// TwinCAT 3 PLC project ValentaDCmotor
// ProgramVersion: 3.1.4026.20
// libraries:
//   Tc2_Standard, * (Beckhoff Automation GmbH)
//   Tc2_System, * (Beckhoff Automation GmbH)
//   Tc3_Module, * (Beckhoff Automation GmbH)
//   VisuDialogs, * (System)
//   VisuSymbols,3.5.10.0,System
// project tree:
//   DUTs/ E_Color.TcDUT, E_ControlMode.TcDUT, E_DoorState.TcDUT, ST_KeyControl.TcDUT, E_BlinkMarine_Color.TcDUT, E_GearState.TcDUT, E_LedColor.TcDUT, E_BacklightColor.TcDUT, E_ValveState.TcDUT, ST_UcWinchControl.TcDUT
//   / GlobalTextList.TcGTLO, PlcTask.TcTTO
//   GVLs/ GVL.TcGVL, GVL_Alarms.TcGVL, GVL_CAN.TcGVL, GVL_ENGINE.TcGVL, GVL_HMI.TcGVL, GVL_IO.TcGVL, GVL_PERSISTENT.TcGVL
//   POUs/ DirectMotorControl.TcPOU, MAIN.TcPOU, PRG_Ballast.TcPOU, PRG_BlinkMarine.TcPOU, PRG_Doors.TcPOU, PRG_Engine.TcPOU, PRG_HmiLeds.TcPOU, PRG_Sequence.TcPOU, PRG_StationManager.TcPOU, PRG_Can.TcPOU, PRG_Winches.TcPOU, PRG_ZF_Control.TcPOU
//   POUs/FBs/ FB_BallastValve.TcPOU, FB_DC_Motor_Direct_Ctrl.TcPOU, FB_DoorControl.TcPOU, FB_EngineControl.TcPOU, FB_StationManager.TcPOU, FB_TankScaling.TcPOU, FB_TunelPump.TcPOU, FB_WinchControl.TcPOU, MeasureRPM.TcPOU
//   POUs/Sim/ E_SystemMode.TcDUT, PRG_SimDoors.TcPOU
//   VISUs/ Visualization1.TcVIS, Visualization2.TcVIS, VisualizationManager.TcVMO (not stored), VisuDoorControl.TcVIS
// real-time tasks:
//   TASK PlcTask: cycle T#2ms, priority 20, ADS port 350
// I/O:
//   DEVICE Device 1 (EtherCAT), AmsNetId 5.168.36.149.2.1
//     Term 1 (EK1200) [EK1200-5000 EtherCAT Power supply (2A E-Bus)]
//       Term 2 (EL1008) [EL1008 8Ch. Dig. Input 24V, 3ms]
//       Term 3 (EL2008) [EL2008 8Ch. Dig. Output 24V, 0.5A]
//       Term 4 (EL4018) [EL4018 8Ch. Ana. Output 0-20mA, 12bit]
//       Term 5 (EL6751) [EL6751 CANopen Master]
//       Term 6 (EK1110) [EK1110 EtherCAT extension]
//     Term 7 (EK1100) [EK1100 EtherCAT Coupler (2A E-Bus)]
//       Term 8 (EL1008) [EL1008 8Ch. Dig. Input 24V, 3ms]
//       Term 9 (EL1008) [EL1008 8Ch. Dig. Input 24V, 3ms]
//       Term 10 (EL1008) [EL1008 8Ch. Dig. Input 24V, 3ms]
//       Term 11 (EL3014) [EL3014 4Ch. Ana. Input 0-20mA DIFF]
//       Term 12 (EL3014) [EL3014 4Ch. Ana. Input 0-20mA DIFF]
//       Term 13 (EL3014) [EL3014 4Ch. Ana. Input 0-20mA DIFF]
//       Term 14 (EL3004) [EL3004 4Ch. Ana. Input +/-10V]
//       Term 15 (EL3255) [EL3255 5Ch. potentiometer measurement with sensor supply]
//       Term 16 (EL7342) [EL7342 2Ch. DC motor output stage (50V, 3.5A)]
//       Term 17 (EL2008) [EL2008 8Ch. Dig. Output 24V, 0.5A]
//       Term 18 (EL2008) [EL2008 8Ch. Dig. Output 24V, 0.5A]
//       Term 19 (EL2008) [EL2008 8Ch. Dig. Output 24V, 0.5A]
//       Term 20 (EL2008) [EL2008 8Ch. Dig. Output 24V, 0.5A]
//       Term 21 (EL9011) [EL9011 End Terminal]
//   DEVICE Device 2 (EL6751), AmsNetId 5.168.36.149.3.1
//     Box 10 (BlinkMarine)
//     Box 11 (BlinkMarine)
//     Box 20 (BlinkMarine)
// variable links:
//   ValentaDCmotor/ValentaDCmotor Instance <-> Device 1 (EtherCAT)/Term 7 (EK1100)/Term 15 (EL3255)
//     PlcTask Inputs/GVL.iwPotFeedback_M1 <-> AI Standard Channel 1/Value
//     PlcTask Inputs/GVL.iwPotFeedback_M2 <-> AI Standard Channel 2/Value
//     PlcTask Inputs/GVL_IO.iLever_St1_Raw <-> AI Standard Channel 3/Value
//     PlcTask Inputs/GVL_IO.iLever_St2_Raw <-> AI Standard Channel 4/Value
//   ValentaDCmotor/ValentaDCmotor Instance <-> Device 1 (EtherCAT)/Term 7 (EK1100)/Term 16 (EL7342)
//     PlcTask Inputs/GVL.bDigitalInput1_M1 <-> DCM Status Channel 1/Status/Digital input 1
//     PlcTask Inputs/GVL.bDigitalInput1_M2 <-> DCM Status Channel 2/Status/Digital input 1
//     PlcTask Inputs/GVL.bDigitalInput2_M1 <-> DCM Status Channel 1/Status/Digital input 2
//     PlcTask Inputs/GVL.bDigitalInput2_M2 <-> DCM Status Channel 2/Status/Digital input 2
//     PlcTask Inputs/GVL.bError_M1 <-> DCM Status Channel 1/Status/Error
//     PlcTask Inputs/GVL.bError_M2 <-> DCM Status Channel 2/Status/Error
//     PlcTask Inputs/GVL.bMovingNegative_M1 <-> DCM Status Channel 1/Status/Moving negative
//     PlcTask Inputs/GVL.bMovingNegative_M2 <-> DCM Status Channel 2/Status/Moving negative
//     PlcTask Inputs/GVL.bMovingPositive_M1 <-> DCM Status Channel 1/Status/Moving positive
//     PlcTask Inputs/GVL.bMovingPositive_M2 <-> DCM Status Channel 2/Status/Moving positive
//     PlcTask Inputs/GVL.bReadyToEnable_M1 <-> DCM Status Channel 1/Status/Ready to enable
//     PlcTask Inputs/GVL.bReadyToEnable_M2 <-> DCM Status Channel 2/Status/Ready to enable
//     PlcTask Inputs/GVL.bReady_M1 <-> DCM Status Channel 1/Status/Ready
//     PlcTask Inputs/GVL.bReady_M2 <-> DCM Status Channel 2/Status/Ready
//     PlcTask Inputs/GVL.bSyncError_M1 <-> DCM Status Channel 1/Status/Sync error
//     PlcTask Inputs/GVL.bSyncError_M2 <-> DCM Status Channel 2/Status/Sync error
//     PlcTask Inputs/GVL.bTorqueReduced_M1 <-> DCM Status Channel 1/Status/Torque reduced
//     PlcTask Inputs/GVL.bTorqueReduced_M2 <-> DCM Status Channel 2/Status/Torque reduced
//     PlcTask Inputs/GVL.bTxPDOToggle_M1 <-> DCM Status Channel 1/Status/TxPDO Toggle
//     PlcTask Inputs/GVL.bTxPDOToggle_M2 <-> DCM Status Channel 2/Status/TxPDO Toggle
//     PlcTask Inputs/GVL.bWarning_M1 <-> DCM Status Channel 1/Status/Warning
//     PlcTask Inputs/GVL.bWarning_M2 <-> DCM Status Channel 2/Status/Warning
//     PlcTask Inputs/GVL.nMotorCurrent_M1 <-> DCM Synchron info data Channel 1/Info data 2
//     PlcTask Inputs/GVL.nMotorCurrent_M2 <-> DCM Synchron info data Channel 2/Info data 2
//     PlcTask Inputs/GVL.nMotorVoltage_M1 <-> DCM Synchron info data Channel 1/Info data 1
//     PlcTask Inputs/GVL.nMotorVoltage_M2 <-> DCM Synchron info data Channel 2/Info data 1
//     PlcTask Outputs/GVL.bEnable_M1 <-> DCM Control Channel 1/Control/Enable
//     PlcTask Outputs/GVL.bEnable_M2 <-> DCM Control Channel 2/Control/Enable
//     PlcTask Outputs/GVL.bReduceTorque_M1 <-> DCM Control Channel 1/Control/Reduce torque
//     PlcTask Outputs/GVL.bReduceTorque_M2 <-> DCM Control Channel 2/Control/Reduce torque
//     PlcTask Outputs/GVL.bReset_M1 <-> DCM Control Channel 1/Control/Reset
//     PlcTask Outputs/GVL.bReset_M2 <-> DCM Control Channel 2/Control/Reset
//     PlcTask Outputs/GVL.nVelocitySetpoint_M1 <-> DCM Velocity Channel 1/Velocity
//     PlcTask Outputs/GVL.nVelocitySetpoint_M2 <-> DCM Velocity Channel 2/Velocity
//   ValentaDCmotor/ValentaDCmotor Instance <-> Device 1 (EtherCAT)/Term 7 (EK1100)/Term 17 (EL2008)
//     PlcTask Outputs/GVL_IO.DO_DoorAft_Close <-> Channel 3/Output
//     PlcTask Outputs/GVL_IO.DO_DoorAft_Open <-> Channel 4/Output
//     PlcTask Outputs/GVL_IO.DO_DoorFwd_Close <-> Channel 1/Output
//     PlcTask Outputs/GVL_IO.DO_DoorFwd_Open <-> Channel 2/Output
//     PlcTask Outputs/GVL_IO.bDcPump_Start <-> Channel 6/Output
//     PlcTask Outputs/GVL_IO.bValve_Winch1_A <-> Channel 7/Output
//     PlcTask Outputs/GVL_IO.bValve_Winch1_B <-> Channel 8/Output
//   ValentaDCmotor/ValentaDCmotor Instance <-> Device 1 (EtherCAT)/Term 7 (EK1100)/Term 18 (EL2008)
//     PlcTask Outputs/GVL_IO.bValve_Winch2_A <-> Channel 1/Output
//     PlcTask Outputs/GVL_IO.bValve_Winch3_A <-> Channel 3/Output
//     PlcTask Outputs/GVL_IO.bValve_Winch2_B <-> Channel 2/Output
//     PlcTask Outputs/GVL_IO.bValve_Winch3_B <-> Channel 4/Output
//   ValentaDCmotor/ValentaDCmotor Instance <-> Device 1 (EtherCAT)/Term 7 (EK1100)/Term 19 (EL2008)
//     PlcTask Outputs/GVL_IO.DO_Engine_Ignition <-> Channel 1/Output
//     PlcTask Outputs/GVL_IO.DO_Engine_Starter <-> Channel 2/Output
//     PlcTask Outputs/GVL_IO.DO_Engine_Stop <-> Channel 3/Output
//     PlcTask Outputs/GVL_IO.DO_TunelClutch <-> Channel 4/Output
//   ValentaDCmotor/ValentaDCmotor Instance <-> Device 1 (EtherCAT)/Term 7 (EK1100)/Term 20 (EL2008)
//     PlcTask Outputs/GVL_IO.DO_BAL_P1 <-> Channel 1/Output
//     PlcTask Outputs/GVL_IO.DO_BAL_P2 <-> Channel 2/Output
//     PlcTask Outputs/GVL_IO.DO_BAL_P3 <-> Channel 3/Output
//     PlcTask Outputs/GVL_IO.DO_BAL_S1 <-> Channel 4/Output
//     PlcTask Outputs/GVL_IO.DO_BAL_S2 <-> Channel 5/Output
//     PlcTask Outputs/GVL_IO.DO_BAL_S3 <-> Channel 6/Output
//     PlcTask Outputs/GVL_IO.DO_SondePower <-> Channel 8/Output
//     PlcTask Outputs/GVL_IO.DO_TUNEL_VALVE <-> Channel 7/Output
//   ValentaDCmotor/ValentaDCmotor Instance <-> Device 2 (EL6751)/Box 10 (BlinkMarine)
//     PlcTask Inputs/GVL_CAN.ID10_KeyState <-> TxPDO 1/Inputs/Key State
//     PlcTask Outputs/GVL_CAN.ID10_LedBlinkBlue <-> RxPDO 2/Outputs/Led Blink State Blue
//     PlcTask Outputs/GVL_CAN.ID10_LedBlinkGreen <-> RxPDO 2/Outputs/Led Blink State Green
//     PlcTask Outputs/GVL_CAN.ID10_LedBlinkRed <-> RxPDO 2/Outputs/Led Blink State Red
//     PlcTask Outputs/GVL_CAN.ID10_LedBlue <-> RxPDO 1/Outputs/Led State Blue
//     PlcTask Outputs/GVL_CAN.ID10_LedGreen <-> RxPDO 1/Outputs/Led State Green
//     PlcTask Outputs/GVL_CAN.ID10_LedRed <-> RxPDO 1/Outputs/Led State Red
//   ValentaDCmotor/ValentaDCmotor Instance <-> Device 2 (EL6751)/Box 11 (BlinkMarine)
//     PlcTask Inputs/GVL_CAN.ID11_KeyState <-> TxPDO 1/Inputs/Key State
//     PlcTask Outputs/GVL_CAN.ID11_LedBlinkBlue <-> RxPDO 2/Outputs/Led Blink State Blue
//     PlcTask Outputs/GVL_CAN.ID11_LedBlinkGreen <-> RxPDO 2/Outputs/Led Blink State Green
//     PlcTask Outputs/GVL_CAN.ID11_LedBlinkRed <-> RxPDO 2/Outputs/Led Blink State Red
//     PlcTask Outputs/GVL_CAN.ID11_LedBlue <-> RxPDO 1/Outputs/Led State Blue
//     PlcTask Outputs/GVL_CAN.ID11_LedGreen <-> RxPDO 1/Outputs/Led State Green
//     PlcTask Outputs/GVL_CAN.ID11_LedRed <-> RxPDO 1/Outputs/Led State Red
//   ValentaDCmotor/ValentaDCmotor Instance <-> Device 2 (EL6751)/Box 20 (BlinkMarine)
//     PlcTask Inputs/GVL_CAN.ID20_KeyState <-> TxPDO 1/Inputs/Key State
//     PlcTask Outputs/GVL_CAN.ID20_LedBlinkBlue <-> RxPDO 2/Outputs/Led Blink State Blue
//     PlcTask Outputs/GVL_CAN.ID20_LedBlinkGreen <-> RxPDO 2/Outputs/Led Blink State Green
//     PlcTask Outputs/GVL_CAN.ID20_LedBlinkRed <-> RxPDO 2/Outputs/Led Blink State Red
//     PlcTask Outputs/GVL_CAN.ID20_LedBlue <-> RxPDO 1/Outputs/Led State Blue
//     PlcTask Outputs/GVL_CAN.ID20_LedGreen <-> RxPDO 1/Outputs/Led State Green
//     PlcTask Outputs/GVL_CAN.ID20_LedRed <-> RxPDO 1/Outputs/Led State Red

CONFIGURATION ValentaDCmotor
    RESOURCE PLC ON TwinCAT3
        TASK PlcTask(INTERVAL := T#2ms, PRIORITY := 20);
        PROGRAM MAIN WITH PlcTask : MAIN;
    END_RESOURCE
END_CONFIGURATION

// ---- DUTs/E_Color.TcDUT
{attribute 'qualified_only'}
{attribute 'strict'}
{attribute 'to_string'}
TYPE E_Color :
(
	eSilver,
	eLime,
	eYellow,
	eOrange,
	eRed,
	eBlue
);
END_TYPE

// ---- DUTs/E_ControlMode.TcDUT
{attribute 'qualified_only'}
{attribute 'strict'}
{attribute 'to_string'}
TYPE E_ControlMode :
(
	OFF  := 0,
	MAN  := 1,
	AUTO := 2
) USINT;
END_TYPE

// ---- DUTs/E_DoorState.TcDUT
{attribute 'qualified_only'}
{attribute 'strict'}
TYPE E_DoorState :
(
    IDLE             := 0,  (* Miruje, nema komande *)
    OPEN             := 1,  (* Potvrđeno otvoreno - održava tlak *)
    CLOSED           := 2,  (* Potvrđeno zatvoreno - održava tlak *)
    TRAVELING_OPEN   := 10, (* Putuje prema otvorenom *)
    TRAVELING_CLOSE  := 20  (* Putuje prema zatvorenom *)
);
END_TYPE

// ---- DUTs/ST_KeyControl.TcDUT
TYPE ST_KeyControl :
STRUCT
    Boja  : E_BlinkMarine_Color; // Koju boju želiš
    Blink : BOOL;                // Želiš li da blica
END_STRUCT
END_TYPE

// ---- DUTs/E_BlinkMarine_Color.TcDUT
{attribute 'qualified_only'}
{attribute 'strict'}
{attribute 'to_string'}
TYPE E_BlinkMarine_Color :
(
    OFF      := 0,
    RED      := 1,
    GREEN    := 2,
    BLUE     := 3,
    YELLOW   := 4,
    CYAN     := 5,
    MAGENTA  := 6,
    WHITE    := 7,
    AMBER    := 8,   // Neki modeli podržavaju dodatne boje
    ORANGE   := 9
) USINT;
END_TYPE

// ---- DUTs/E_GearState.TcDUT
{attribute 'qualified_only'}
{attribute 'strict'}
TYPE E_GearState :
(
    GEAR_NEUTRAL := 0,
    GEAR_FWD     := 1,
    GEAR_REV     := 2
);
END_TYPE

// ---- DUTs/E_LedColor.TcDUT
{attribute 'qualified_only'}
{attribute 'strict'}
{attribute 'to_string'}
TYPE E_LedColor :
(
    Off := 0,
    Red := 1,
    Green := 2,
    Blue := 3,
    Yellow := 4,
    Cyan := 5,
    Magenta := 6,
    White := 7
) USINT := Off;
END_TYPE

// ---- DUTs/E_BacklightColor.TcDUT
{attribute 'qualified_only'}
{attribute 'strict'}
{attribute 'to_string'}
TYPE E_BacklightColor :
(
    Red := 1,
    Green := 2,
    Blue := 3,
    Yellow := 4,
    Cyan := 5,
    Violet := 6,
    White := 7,
    Amber := 8,
    YellowGreen := 9
) USINT := Amber;
END_TYPE

// ---- DUTs/E_ValveState.TcDUT
{attribute 'qualified_only'}
{attribute 'strict'}
TYPE E_ValveState :
(
    VALVE_UNKNOWN := 0,      (* Ni otvoren ni zatvoren - putuje *)
    VALVE_OPEN := 1,         (* Potvrđeno otvoren *)
    VALVE_CLOSED := 2,       (* Potvrđeno zatvoren *)
    VALVE_ERROR := 3         (* Greška: timeout ili oba signala aktivna *)
);
END_TYPE

// ---- DUTs/ST_UcWinchControl.TcDUT
TYPE ST_UcWinchControl :
STRUCT
    bDisable          : BOOL; (* Glavni Safety Enable *)
    bManualEnable     : BOOL; (* HMI Manual Mode *)
    bBtn_Dir1         : BOOL; (* Tipka: Slow ili In *)
    bBtn_Dir2         : BOOL; (* Tipka: Fast ili Out *)
    bValve_Dir1       : BOOL; (* Aktivan izlaz 1 *)
    bValve_Dir2       : BOOL; (* Aktivan izlaz 2 *)
    bReq_Pump         : BOOL; (* Pumpa radi *)
    bSts_SystemSafe   : BOOL; (* Zeleno = Safe *)
    bSts_ManualEn     : BOOL; (* Zeleno = Manual *)
END_STRUCT
END_TYPE

// ---- POUs/Sim/E_SystemMode.TcDUT
{attribute 'qualified_only'}
{attribute 'strict'}
TYPE E_SystemMode :
(
    MODE_IDLE   := 0,  (* Sustav miruje / Inicijalizacija *)
    MODE_DRIVE  := 1,  (* POGON: Oba vrata otvorena *)
    MODE_SAIL   := 2,  (* JEDRENJE: Prednja otvorena, Zadnja zatvorena *)
    MODE_ERROR  := 3   (* Greška sustava *)
);
END_TYPE

// ---- GVLs/GVL.TcGVL
VAR_GLOBAL

// MOTOR1 ==============
//  Potenciometar feedback EL3255
	iwPotFeedback_M1 AT %I*: INT;	// AI Channel 1

// nControlWord bitovi
	bEnable_M1 AT %Q*: BOOL;         // DCM Control Channel 1.Enable
	bReset_M1 AT %Q*: BOOL;          // DCM Control Channel 1.Reset  
	bReduceTorque_M1 AT %Q*: BOOL;   // DCM Control Channel 1.Reduce torque

    nVelocitySetpoint_M1 AT %Q*: INT; // Link na "Velocity" (49.0)
		
// DCM Status Channel 1 - Input bitovi Link na "Status" (45.0)
	bReadyToEnable_M1 AT %I*: BOOL;    // Spreman za enable
	bReady_M1 AT %I*: BOOL;             // Općenito spreman
	bWarning_M1 AT %I*: BOOL;           // Upozorenje aktivno
	bError_M1 AT %I*: BOOL;             // Greška aktivna
	bMovingPositive_M1 AT %I*: BOOL;    // Kreće se u + smjeru
	bMovingNegative_M1 AT %I*: BOOL;    // Kreće se u - smjeru  
	bTorqueReduced_M1 AT %I*: BOOL;     // Reduce torque aktivan
	bDigitalInput1_M1 AT %I*: BOOL;     // Digitalni ulaz 1
	bDigitalInput2_M1 AT %I*: BOOL;     // Digitalni ulaz 2
	bSyncError_M1 AT %I*: BOOL;         // Sync greška
	bTxPDOToggle_M1 AT %I*: BOOL;       // PDO toggle bit	
	
// Novo - Info data
    nMotorVoltage_M1 AT %I*: UINT; // Info data 1 (mV)
    nMotorCurrent_M1 AT %I*: UINT; // Info data 2 (mA)
	
// MOTOR2 ==============
//  Potenciometar feedback EL3255
	iwPotFeedback_M2 AT %I*: INT;	// AI Channel 1

// nControlWord bitovi
	bEnable_M2 AT %Q*: BOOL;         // DCM Control Channel 1.Enable
	bReset_M2 AT %Q*: BOOL;          // DCM Control Channel 1.Reset  
	bReduceTorque_M2 AT %Q*: BOOL;   // DCM Control Channel 1.Reduce torque

    nVelocitySetpoint_M2 AT %Q*: INT; // Link na "Velocity" (49.0)
		
// DCM Status Channel 1 - Input bitovi Link na "Status" (45.0)
	bReadyToEnable_M2 AT %I*: BOOL;    // Spreman za enable
	bReady_M2 AT %I*: BOOL;             // Općenito spreman
	bWarning_M2 AT %I*: BOOL;           // Upozorenje aktivno
	bError_M2 AT %I*: BOOL;             // Greška aktivna
	bMovingPositive_M2 AT %I*: BOOL;    // Kreće se u + smjeru
	bMovingNegative_M2 AT %I*: BOOL;    // Kreće se u - smjeru  
	bTorqueReduced_M2 AT %I*: BOOL;     // Reduce torque aktivan
	bDigitalInput1_M2 AT %I*: BOOL;     // Digitalni ulaz 1
	bDigitalInput2_M2 AT %I*: BOOL;     // Digitalni ulaz 2
	bSyncError_M2 AT %I*: BOOL;         // Sync greška
	bTxPDOToggle_M2 AT %I*: BOOL;       // PDO toggle bit	
	
// Novo - Info data
    nMotorVoltage_M2 AT %I*: UINT; // Info data 1 (mV)
    nMotorCurrent_M2 AT %I*: UINT; // Info data 2 (mA)
	
	
	
END_VAR

// ---- GVLs/GVL_Alarms.TcGVL
{attribute 'qualified_only'}
VAR_GLOBAL
    bAnyAlarmActive : BOOL; (* Zbirni alarm *)
	bErr_DoorFwd : BOOL;
	bLeak_DoorFwd : BOOL;
	bErr_DoorAft : BOOL;
	bLeak_DoorAft : BOOL;
	
END_VAR

// ---- GVLs/GVL_CAN.TcGVL
VAR_GLOBAL
	// --- ID10 (4 tipke) ---
	ID10_KeyState AT %I* : USINT;
	ID10_LedRed AT %Q* : USINT;
	ID10_LedGreen AT %Q* : USINT;
	ID10_LedBlue AT %Q* : USINT;
	ID10_LedBlinkRed AT %Q* : USINT;
	ID10_LedBlinkGreen AT %Q* : USINT;
	ID10_LedBlinkBlue AT %Q* : USINT;
	
	ID10_Config : ARRAY[1..4] OF ST_KeyControl; // Za upisivanje boje i blinka
	ID10_Status : ARRAY[1..4] OF BOOL;          // Za čitanje pritiska tipke

	// --- ID11 (4 tipke) ---
	ID11_KeyState AT %I* : USINT;
	ID11_LedRed AT %Q* : USINT;
	ID11_LedGreen AT %Q* : USINT;
	ID11_LedBlue AT %Q* : USINT;
	ID11_LedBlinkRed AT %Q* : USINT;
	ID11_LedBlinkGreen AT %Q* : USINT;
	ID11_LedBlinkBlue AT %Q* : USINT;
	
	ID11_Config : ARRAY[1..4] OF ST_KeyControl;
	ID11_Status : ARRAY[1..4] OF BOOL;

	// --- ID20 (15 tipki) ---
	ID20_KeyState AT %I* : UINT;
	ID20_LedRed AT %Q* : UINT;
	ID20_LedGreen AT %Q* : UINT;
	ID20_LedBlue AT %Q* : UINT;
	ID20_LedBlinkRed AT %Q* : UINT;
	ID20_LedBlinkGreen AT %Q* : UINT;
	ID20_LedBlinkBlue AT %Q* : UINT;
	
	ID20_Config : ARRAY[1..15] OF ST_KeyControl;
	ID20_Status : ARRAY[1..15] OF BOOL;
END_VAR

// ---- GVLs/GVL_ENGINE.TcGVL
{attribute 'qualified_only'}
VAR_GLOBAL
    fEngineRPM      : REAL;
    fThrottleOut    : REAL;
    eGearOut        : E_GearState;
    bIsShifting     : BOOL;
    bAlarm_HighRPM  : BOOL;
	
	(* Triggeri za tipke *)
    rtStart_ID10, rtStart_ID11 : R_TRIG;
    rtStop_ID10,  rtStop_ID11  : R_TRIG;
    rtSel_ID10,   rtSel_ID11   : R_TRIG;

    (* Timeri za sekvence *)
    tmrStopSequence : TON;
    
    (* Interne statusne varijable *)
    bIgnitionActive : BOOL; 
    bEngineRunning  : BOOL;
    iActiveStation  : INT := 1; // 1 = Port (ID10), 2 = Stbd (ID11)
END_VAR

// ---- GVLs/GVL_HMI.TcGVL
{attribute 'qualified_only'}
VAR_GLOBAL
    (* --- KOMANDE SA EKRANA (Tipke) --- *)
    (* TRUE = Operater želi otvoriti ventil *)
	eSystemMode : E_ControlMode := E_ControlMode.OFF;
    bCmdOpen_P : ARRAY[1..3] OF BOOL; // Komande za Port
    bCmdOpen_S : ARRAY[1..3] OF BOOL; // Komande za Stbd
	
    bCmdOpen_P1 : BOOL;
    bCmdOpen_P2 : BOOL;
    bCmdOpen_P3 : BOOL;
    bCmdOpen_S1 : BOOL;
    bCmdOpen_S2 : BOOL;
    bCmdOpen_S3 : BOOL;
    bCmdOpen_Tunel : BOOL;
    
    (* Reset tipka za alarme *)
    bCmdResetAll : BOOL;

    (* --- STATUSI ZA EKRAN (Boje/Tekst) --- *)
    (* Koristimo onaj ENUM koji smo napravili: 1=Open, 2=Closed... *)
    eState_P1 : E_ValveState;
    eState_P2 : E_ValveState;
    eState_P3 : E_ValveState;
    eState_S1 : E_ValveState;
    eState_S2 : E_ValveState;
    eState_S3 : E_ValveState;
    eState_Tunel : E_ValveState;

    (* --- ALARMI ZA EKRAN (Crvena lampica) --- *)
    bAlarm_P1 : BOOL;
    bAlarm_P2 : BOOL;
    bAlarm_P3 : BOOL;
    bAlarm_S1 : BOOL;
    bAlarm_S2 : BOOL;
    bAlarm_S3 : BOOL;
    bAlarm_Tunel : BOOL;
	
	(* --- VRATA --- *)
    bCmdDoorFwd  : BOOL;
    bCmdDoorAft  : BOOL;
    bCmdDoorFwd_Open  : BOOL;
    bCmdDoorFwd_Close : BOOL;
    bCmdDoorAft_Open  : BOOL;
    bCmdDoorAft_Close : BOOL;

    eState_DoorFwd    : INT; (* Koristimo isti enum: 1=Open, 2=Closed *)
    eState_DoorAft    : INT;
    
    bAlarm_DoorFwd    : BOOL;
    bAlarm_DoorAft    : BOOL;	
	
	(* --- TUNEL PUMP --- *)
	bCmdRun_TunelPump	: BOOL;
	
    (* --- KONFIGURACIJA I OPCIJE --- *)
    bConfig_HydraulicBoost : BOOL := FALSE; (* TRUE = PTO i DC rade ZAJEDNO za wincheve *)
	bConfig_AllowPtoInDrive : BOOL := FALSE; (* TRUE = Dozvoli korištenje motorne hidraulike dok vozimo *)
    bConfig_AutoDcBackup    : BOOL := TRUE;  (* TRUE = Ako motor ima premalo okretaja, automatski upali DC pumpu *)
    
    (* Statusi *)
    bHydraulicsSourceEngine : BOOL; (* Motorna pumpa je aktivna *)
    bHydraulicsSourceDC     : BOOL; (* DC pumpa je aktivna *)

	fHandThrottle : REAL;         // Ručica gasa (0-100)
    eGearCommand  : E_GearState;  // Komanda mjenjača (FWD/N/REV)

	bModeSail : BOOL;
	
	(* --- ODABIR MODA (Zahtjev operatera) --- *)
    bReq_ModeDrive : BOOL; (* Tipka: Želim Pogon *)
    bReq_ModeSail  : BOOL; (* Tipka: Želim Jedrenje *)
    bReq_Stop      : BOOL; (* Tipka: STOP / Standby *)

    (* --- TRENUTNI AKTIVNI MOD (Povratna info) --- *)
    eActiveMode    : E_SystemMode; 
    
    (* Statusi sekvence *)
    bSequenceReady : BOOL; (* Spremni za rad (Vrata su u poziciji) *)
	
	bCmdResetAlarms : BOOL;

	test : BOOL;

    (* --- HMI LED STATUSI (postavljaju se u PRG_HmiLeds) --- *)
    (* Ventili - 4 boje: Cyan=Otvoren, Green=Zatvoren, Orange(Yellow)=Putuje, Red=Greška *)
    bLed_P1_Cyan   : BOOL; bLed_P1_Yellow : BOOL; bLed_P1_Red : BOOL; bLed_P1_Green : BOOL;
    bLed_P2_Cyan   : BOOL; bLed_P2_Yellow : BOOL; bLed_P2_Red : BOOL; bLed_P2_Green : BOOL;
    bLed_P3_Cyan   : BOOL; bLed_P3_Yellow : BOOL; bLed_P3_Red : BOOL; bLed_P3_Green : BOOL;
    bLed_S1_Cyan   : BOOL; bLed_S1_Yellow : BOOL; bLed_S1_Red : BOOL; bLed_S1_Green : BOOL;
    bLed_S2_Cyan   : BOOL; bLed_S2_Yellow : BOOL; bLed_S2_Red : BOOL; bLed_S2_Green : BOOL;
    bLed_S3_Cyan   : BOOL; bLed_S3_Yellow : BOOL; bLed_S3_Red : BOOL; bLed_S3_Green : BOOL;
    bLed_Tunel_Cyan   : BOOL; bLed_Tunel_Yellow : BOOL; bLed_Tunel_Red : BOOL; bLed_Tunel_Green : BOOL;
    (* Pumpa *)
    bLed_Pump_Cyan : BOOL; bLed_Pump_Red  : BOOL;
    (* Motor *)
    bLed_Engine_Green : BOOL;
    (* Vrata *)
    bLed_DoorFwd_Cyan : BOOL; bLed_DoorFwd_Yellow : BOOL; bLed_DoorFwd_Red : BOOL; bLed_DoorFwd_Green : BOOL;
    bLed_DoorAft_Cyan : BOOL; bLed_DoorAft_Yellow : BOOL; bLed_DoorAft_Red : BOOL; bLed_DoorAft_Green : BOOL;

END_VAR

// ---- GVLs/GVL_IO.TcGVL
{attribute 'qualified_only'}
VAR_GLOBAL
    (* --- DIGITALNI ULAZI (Feedback sa ventila) --- *)

    (* --- SIGURNOSNI PREKIDAČI (NC - Normalno Zatvoreni) --- *)
    (* TRUE = OK, FALSE = Pritisnut/prekinut = STOP *)
    DI_Stop_Port   AT %I* : BOOL; (* NC Stop tipka Port strana *)
    DI_Stop_Stbd   AT %I* : BOOL; (* NC Stop tipka Starboard strana *)

    (* PORT Strana *)
    DI_BAL_P1_OPEN_FB   AT %I* : BOOL;
    DI_BAL_P1_CLOSE_FB  AT %I* : BOOL;
    DI_BAL_P2_OPEN_FB   AT %I* : BOOL;
    DI_BAL_P2_CLOSE_FB  AT %I* : BOOL;
    DI_BAL_P3_OPEN_FB   AT %I* : BOOL;
    DI_BAL_P3_CLOSE_FB  AT %I* : BOOL;

    (* STARBOARD Strana *)
    DI_BAL_S1_OPEN_FB   AT %I* : BOOL;
    DI_BAL_S1_CLOSE_FB  AT %I* : BOOL;
    DI_BAL_S2_OPEN_FB   AT %I* : BOOL;
    DI_BAL_S2_CLOSE_FB  AT %I* : BOOL;
    DI_BAL_S3_OPEN_FB   AT %I* : BOOL;
    DI_BAL_S3_CLOSE_FB  AT %I* : BOOL;

    (* --- NOVO: TUNEL PUMP (Ventil za usmjeravanje) --- *)
    DI_TUNEL_OPEN_FB    AT %I* : BOOL;
    DI_TUNEL_CLOSE_FB   AT %I* : BOOL;
	// --- NOVO: TUNEL PUMP HARDWARE ---
	DI_Sonda_Port        AT %I* : BOOL; // Senzor u Port usisu
    DI_Sonda_Stbd        AT %I* : BOOL; // Senzor u Stbd usisu
    DO_TunelClutch       AT %Q* : BOOL; // Izlaz za uključivanje kuplunga pumpe
    DO_SondePower		 AT %Q* : BOOL; // Zajedničko napajanje za obje sonde (0.5A)
	
    (* --- DIGITALNI IZLAZI --- *)
    (* PORT Strana *)
    DO_BAL_P1           AT %Q* : BOOL;
    DO_BAL_P2           AT %Q* : BOOL;
    DO_BAL_P3           AT %Q* : BOOL;

    (* STARBOARD Strana *)
    DO_BAL_S1           AT %Q* : BOOL;
    DO_BAL_S2           AT %Q* : BOOL;
    DO_BAL_S3           AT %Q* : BOOL;

    (* --- NOVO: TUNEL PUMP IZLAZ --- *)
    DO_TUNEL_VALVE      AT %Q* : BOOL;
	
    (* --- VRATA (Hidraulika) --- *)
    (* Digitalni Izlazi (24V Špule) *)
    DO_DoorFwd_Open    AT %Q* : BOOL;
    DO_DoorFwd_Close   AT %Q* : BOOL;
    
    DO_DoorAft_Open    AT %Q* : BOOL;
    DO_DoorAft_Close   AT %Q* : BOOL;
	
    (* --- ULAZI (TIPKE NA PALUBI) --- *)
    (* Svaki vinč ima 2 gumba (npr. Brzina 1 / Brzina 2 ili Trim / Ease) *)
    bBtn_Winch1_A  AT %I* : BOOL;
    bBtn_Winch1_B  AT %I* : BOOL;
    
    bBtn_Winch2_A  AT %I* : BOOL;
    bBtn_Winch2_B  AT %I* : BOOL;
    
    bBtn_Winch3_A  AT %I* : BOOL;
    bBtn_Winch3_B  AT %I* : BOOL;

    (* --- IZLAZI (HIDRAULIČKI VENTILI) --- *)
    bValve_Winch1_A AT %Q* : BOOL;
    bValve_Winch1_B AT %Q* : BOOL;
    
    bValve_Winch2_A AT %Q* : BOOL;
    bValve_Winch2_B AT %Q* : BOOL;
    
    bValve_Winch3_A AT %Q* : BOOL;
    bValve_Winch3_B AT %Q* : BOOL;
    
    (* --- DC PUMPA (BACKUP) --- *)
    bDcPump_Start   AT %Q* : BOOL; (* Relej za paljenje DC pumpe *)
    
    (* --- KOMUNIKACIJA S MOTOROM --- *)
    iRpmReq_Winches : INT; (* Koliko RPM-a tražimo od motora *)
    bAnyWinchActive : BOOL; (* Barem jedan radi *)

    (* Analogni Ulazi (Tlak - 4-20mA skalirano u Bar) *)
    fPressure_FWD_A     : REAL; 
    fPressure_FWD_B     : REAL;
    fPressure_AFT_A     : REAL;
    fPressure_AFT_B     : REAL;	
	
    fEngineRPM_Scaled   : REAL;
	
    (* --- ANALOGNI ULAZI (RAW 0..32767) --- *)
    (* Tlakovi Vrata *)
    iPressure_FWD_A_Raw : INT;
    iPressure_FWD_B_Raw : INT;
    iPressure_AFT_A_Raw : INT;
    iPressure_AFT_B_Raw : INT;

    (* ZF Aktuator Feedback *)
    iGas_ActualPos_Raw  AT %I* : INT;
    iGear_ActualPos_Raw AT %I* : INT;
    
    (* Ručice (Komande) *)
    iLever_St1_Raw      AT %I* : INT; (* Komanda Stanica 1 *)
    iLever_St2_Raw      AT %I* : INT; (* Komanda Stanica 2 *)
    iActiveLever_Raw    : INT; (* Odabrana ručica koja ide na motor *)
    
    (* --- DIGITALNI SIGNALI (Station Manager) --- *)
    bBtn_Sel_St1        : BOOL;
    bLed_Sel_St1        : BOOL;
    bBtn_Sel_St2        : BOOL;
    bLed_Sel_St2        : BOOL;
    bBuzzer             : BOOL;

    (* --- IZLAZI ZA EL7342 (ZF Aktuator) --- *)
    nGas_Motor_Out      : INT;
    nGear_Motor_Out     : INT;
	
    (* --- BALASTI (6 TANKOVA) - ULAZI 4-20mA --- *)
    (* Lijeva strana (PORT) *)
    iLevel_Bal_P1_Raw   AT %I* : INT; (* Port 1 (Pramac/Forward) *)
    iLevel_Bal_P2_Raw   AT %I* : INT; (* Port 2 (Mid) *)
    iLevel_Bal_P3_Raw   AT %I* : INT; (* Port 3 (Krma/Aft) *)
    
    (* Desna strana (STARBOARD) *)
    iLevel_Bal_S1_Raw   AT %I* : INT; (* Stbd 1 *)
    iLevel_Bal_S2_Raw   AT %I* : INT; (* Stbd 2 *)
    iLevel_Bal_S3_Raw   AT %I* : INT; (* Stbd 3 *)

    (* --- SKALIRANE VRIJEDNOSTI (0.0 - 100.0 %) --- *)
    (* PORT *)
    fLevel_Bal_P1_Pct_Hmi   : REAL;
    fLevel_Bal_P2_Pct_Hmi   : REAL;
    fLevel_Bal_P3_Pct_Hmi   : REAL;
    (* STBD *)
    fLevel_Bal_S1_Pct_Hmi   : REAL;
    fLevel_Bal_S2_Pct_Hmi   : REAL;
    fLevel_Bal_S3_Pct_Hmi   : REAL;
	
	(* PORT *)
    fLevel_Bal_P1_Pct_Disp   AT %Q* : INT;
    fLevel_Bal_P2_Pct_Disp   AT %Q* : INT;
    fLevel_Bal_P3_Pct_Disp   AT %Q* : INT;
    (* STBD *)
    fLevel_Bal_S1_Pct_Disp   AT %Q* : INT;
    fLevel_Bal_S2_Pct_Disp   AT %Q* : INT;
    fLevel_Bal_S3_Pct_Disp   AT %Q* : INT;
    
	(* --- ENGINE --- *)
	DO_Engine_Ignition		AT %Q* : BOOL;
    DO_Engine_Starter		AT %Q* : BOOL;
    DO_Engine_Stop			AT %Q* : BOOL;
	
    (* --- ALARMI --- *)
    bAlarm_HydraulicLow     : BOOL;
    bAlarm_FuelLow          : BOOL;
END_VAR

// ---- GVLs/GVL_PERSISTENT.TcGVL
{attribute 'qualified_only'}
VAR_GLOBAL PERSISTENT
    (* --- KALIBRACIJA RUČICE (INPUT LEVER) --- *)
    (* Ovo su vrijednosti koje očitavaš s pulta (EL3255 Channel 3) *)
    
    iLever_MaxRev    	: INT := 500;   (* Pun gas nazad *)
	iLever_RevGasStart  : INT := 12000;  (* do ove vrijednosti kreće gas u REV *)
    iLever_MinRev    	: INT := 14000;  (* Klik nazad (Početak gasa) *)
   	iLever_RevReturn 	: INT := 15000;  (* povrat iz REV prema neutralu *)
                     	
    iLever_Neutral   	: INT := 16000;  (* Čista sredina *)
                     	
	iLever_FwdReturn 	: INT := 17100;  (* povrat iz FWD prema neutralu *)
    iLever_MinFwd    	: INT := 18100;  (* Klik naprijed (Početak gasa) *)
	iLever_FwdGasStart  : INT := 20500;  (* od ove vrijednosti kreće gas u FWD *)
	iLever_MaxFwd    	: INT := 31500;  (* Pun gas naprijed *)
                     	
    (* --- KALIBRACIJA IZLAZNIH AKTUATORA (MOTOR I KOPČA) --- *)
    (* Ovo su granice motora u kutiji (EL3255 Ch 1 i 2) *)
    
    (* Output Gas (Sajla gasa) *)
    iAct_Gas_Idle   : INT := 10;   (* Fizički minimum sajle *)
    iAct_Gas_Max    : INT := 90;  (* Fizički maksimum sajle *)
    
    (* Output Kopča (Sajla mjenjača) *)
    iAct_Gear_Rev   : INT := 10;
    iAct_Gear_Neut  : INT := 50;
    iAct_Gear_Fwd   : INT := 90;
END_VAR

// ---- POUs/MAIN.TcPOU
PROGRAM MAIN
VAR

END_VAR


PRG_ZF_Control();
PRG_Engine();
PRG_BlinkMarine();
PRG_Ballast();
PRG_Doors();
PRG_Winches();
PRG_SimDoors();
PRG_HmiLeds();

END_PROGRAM

// ---- POUs/PRG_ZF_Control.TcPOU
PROGRAM PRG_ZF_Control
VAR
    (* --- SERVO DRIVERI --- *)
//    fbServoGas  : FB_DC_Servo_PWM;
//    fbServoGear : FB_DC_Servo_PWM;
    
    (* --- INTERNE VARIJABLE --- *)
    fInputRaw   : REAL; (* Pozicija ručice *)
    fGasRequest : REAL; (* Izračunati gas (0.0 - 1.0) *)
    fRange      : REAL; (* Pomoćna za matematiku *)
    
    (* --- CILJEVI (TARGETS) --- *)
    iTargetGas  : INT;
    iTargetGear : INT;
    
    (* --- STATUSI --- *)
   bGearIsSafe : BOOL; (* Kopča je na mjestu *)
    
    (* --- KONVERZIJA RPM ZA VINČEVE --- *)
    fWinchRpmFactor : REAL := 10.0; (* Koliko 'Raw' bodova po 1 RPM-u? Podesi ovo! *)
	
	iGearState : INT := 0;   // -1 = REV, 0 = NEUT, 1 = FWD
	
	RPM_Motor: MeasureRPM;

// Za simulaciju kretanja
	Tgen1: TON;
	bTick1: BOOL;
	R_Tgen1: R_TRIG;
	bTakt1: BOOL;
	bMove_M1: BOOL;	// Sim Move enable
	
	Tgen2: TON;
	bTick2: BOOL;
	R_Tgen2: R_TRIG;
	bTakt2: BOOL;
	bMove_M2: BOOL;	// Sim Move enable

	rSetpointTarget_MinM1: REAL:=22.0;		// Simulacija Targget pos Min
	rSetpointTarget_MaxM1: REAL:=77.0;		// Simulacija Targget pos Max
	rSetpointTarget_MinM2: REAL:=22.0;		// Simulacija Targget pos Min
	rSetpointTarget_MaxM2: REAL:=77.0;		// Simulacija Targget pos Max

// MOTOR_1	
	FB_DC_MOTOR1: FB_DC_Motor_Direct_Ctrl;	// FB DC Motor Ctrl
	// komande
	bMotorOn_M1: BOOL:=TRUE;				// Motor ON
	rSetpointTarget_M1: REAL;		// Setpopoint Target pos percent	
	rMaxVelocityM1: REAL:=100.0;	// Zadana brzina %
	// Parametri
	rKp_M1: REAL:=5.0;	// ostali su fiksni na FB-u
	
	bInDeadband_M1: BOOL;			// u podrucju prozora pozicije
	bHMI_RESET_M1: BOOL;			// reset greske ih HMI
	rErrorM1: LREAL;				// Greska slijedenja pozicije
	bSetVelOverPozM1: BOOL;			// greska set pos koji premasuje INT  - iskljucije Motor
	bSetVelOverNegM1: BOOL;			// greska set pos koji premasuje INT  - iskljucije Motor
	rPotFeedback_Radno_PercM1: REAL;//Pozicija % radnog pomaka 0--100%
	rMotorVoltageM1: REAL;			// monitoring napon motora V
	rMotorCurrentM1: REAL;			// monitoring struja motora A
	rActualVelocityRPM_M1: REAL;	// trnutna brzina motora RPM
	bErrorLimitPosMin_M1: BOOL;	// Pozicija ispod min limita 
	bErrorLimitPosMax_M1: BOOL;	// Pozicija iznad max limita 
	bERROR_COM_M1: BOOL;			// generalna greska
	bERROR_POS_M1: BOOL;			// greska pozicije ako je van pozicije > n sec 
	

// MOTOR_2	
	FB_DC_MOTOR2: FB_DC_Motor_Direct_Ctrl;	// FB DC Motor Ctrl
	// komande
	bMotorOn_M2: BOOL:=true;				// Motor ON
	rSetpointTarget_M2: REAL;		// Setpopoint Target pos percent	
	rMaxVelocityM2: REAL:=100.0;	// Zadana brzina %
	// Parametri
	rKp_M2: REAL:=5.0;	// ostali su fiksni na FB-u
	
	bInDeadband_M2: BOOL;			// u podrucju prozora pozicije
	bHMI_RESET_M2: BOOL;			// reset greske ih HMI
	rErrorM2: LREAL;				// Greska slijedenja pozicije
	bSetVelOverPozM2: BOOL;			// greska set pos koji premasuje INT  - iskljucije Motor
	bSetVelOverNegM2: BOOL;			// greska set pos koji premasuje INT  - iskljucije Motor
	rPotFeedback_Radno_PercM2: REAL;//Pozicija % radnog pomaka 0--100%
	rMotorVoltageM2: REAL;			// monitoring napon motora V
	rMotorCurrentM2: REAL;			// monitoring struja motora A
	rActualVelocityRPM_M2: REAL;	// trnutna brzina motora RPM
	bErrorLimitPosMin_M2: BOOL;	// Pozicija ispod min limita 
	bErrorLimitPosMax_M2: BOOL;	// Pozicija iznad max limita 
	bERROR_COM_M2: BOOL;			// generalna greska
	bERROR_POS_M2: BOOL;			// greska pozicije ako je van pozicije > n sec 
	

	
END_VAR

// =========================================================
// 1. OČITAVANJE ULAZA
// =========================================================
fInputRaw := INT_TO_REAL(GVL_IO.iActiveLever_Raw);


// =========================================================
// 2. LOGIKA KOPČE I GASA IZ RUČICE (S HISTERESISOM)
// =========================================================

// iGearState:
//  -1 = REV
//   0 = NEUT
//   1 = FWD

CASE iGearState OF

    0: // NEUTRAL
        IF fInputRaw >= INT_TO_REAL(GVL_PERSISTENT.iLever_MinFwd) THEN
            iGearState := 1;   // FWD
        ELSIF fInputRaw <= INT_TO_REAL(GVL_PERSISTENT.iLever_MinRev) THEN
            iGearState := -1;  // REV
        END_IF

    1: // FWD
        IF fInputRaw < INT_TO_REAL(GVL_PERSISTENT.iLever_FwdReturn) THEN
            iGearState := 0;   // povrat u neutral
        END_IF

    -1: // REV
        IF fInputRaw > INT_TO_REAL(GVL_PERSISTENT.iLever_RevReturn) THEN
            iGearState := 0;   // povrat u neutral
        END_IF

ELSE
    iGearState := 0;
END_CASE


// Izračun target gear + gas request prema stanju
CASE iGearState OF

    1: // FWD
        iTargetGear := GVL_PERSISTENT.iAct_Gear_Fwd;

        // Gas počinje tek nakon zone izlaska kuglice / detenta
        IF fInputRaw >= INT_TO_REAL(GVL_PERSISTENT.iLever_FwdGasStart) THEN
            fRange := INT_TO_REAL(GVL_PERSISTENT.iLever_MaxFwd - GVL_PERSISTENT.iLever_FwdGasStart);
            IF fRange > 0.0 THEN
                fGasRequest := (fInputRaw - INT_TO_REAL(GVL_PERSISTENT.iLever_FwdGasStart)) / fRange;
            ELSE
                fGasRequest := 0.0;
            END_IF
        ELSE
            fGasRequest := 0.0;
        END_IF

    -1: // REV
        iTargetGear := GVL_PERSISTENT.iAct_Gear_Rev;

        // Gas počinje tek nakon zone izlaska kuglice / detenta
        IF fInputRaw <= INT_TO_REAL(GVL_PERSISTENT.iLever_RevGasStart) THEN
            fRange := INT_TO_REAL(GVL_PERSISTENT.iLever_RevGasStart - GVL_PERSISTENT.iLever_MaxRev);
            IF fRange > 0.0 THEN
                fGasRequest := (INT_TO_REAL(GVL_PERSISTENT.iLever_RevGasStart) - fInputRaw) / fRange;
            ELSE
                fGasRequest := 0.0;
            END_IF
        ELSE
            fGasRequest := 0.0;
        END_IF

ELSE // NEUT
    iTargetGear := GVL_PERSISTENT.iAct_Gear_Neut;
    fGasRequest := 0.0;
END_CASE
// =========================================================
// 3. LIMITIRANJE MATEMATIKE
// =========================================================
IF fGasRequest > 1.0 THEN fGasRequest := 1.0; END_IF
IF fGasRequest < 0.0 THEN fGasRequest := 0.0; END_IF


// =========================================================
// 4. KOMBINIRANJE GASA (POGON vs. VINČEVI)
// =========================================================

// A) AKO VOZIMO (Kopča nije u leru)
IF (iTargetGear <> GVL_PERSISTENT.iAct_Gear_Neut) THEN
    
    // Računamo stvarni položaj aktuatora na temelju ručice
    iTargetGas := REAL_TO_INT(
        fGasRequest * INT_TO_REAL(GVL_PERSISTENT.iAct_Gas_Max - GVL_PERSISTENT.iAct_Gas_Idle)
    ) + GVL_PERSISTENT.iAct_Gas_Idle;

// B) AKO SMO U LERU, A VINČEVI TRAŽE SNAGU
ELSIF (GVL_IO.iRpmReq_Winches > 0) THEN
    
    // Pretvaramo traženi RPM (npr. 1200) u pomak aktuatora
    // Formula: (TraženiRPM - LerRPM) * Faktor + PozicijaLera
    // Podesi 'fWinchRpmFactor' dok ne dobiješ točne okretaje na motoru!
    
    iTargetGas := REAL_TO_INT( (INT_TO_REAL(GVL_IO.iRpmReq_Winches - 700) * fWinchRpmFactor) ) 
                  + GVL_PERSISTENT.iAct_Gas_Idle;
                  
    // Sigurnosni limit da vinčevi ne zakucaju gas do daske
    IF iTargetGas > GVL_PERSISTENT.iAct_Gas_Max THEN 
        iTargetGas := GVL_PERSISTENT.iAct_Gas_Max; 
    END_IF

// C) ČISTI LER
ELSE
    iTargetGas := GVL_PERSISTENT.iAct_Gas_Idle;
END_IF


// =========================================================
// Potenciometar feedback

RPM_Motor(nPotValue:=iwPotFeedback_M1 , nPotValueCount=> , RPM=> );

// DirectMotorControl
// Simulator Reverziranje Motor1 kad uđe u poziciju 
Tgen1(IN:=bInDeadband_M1 , PT:=T#2S , Q=> , ET=> );
R_Tgen1(CLK:=Tgen1.Q , Q=>bTick1 );
IF bTick1 THEN
	bTakt1:=NOT bTakt1;
END_IF
// reverziranje pozicije M1
IF bTakt1 AND bMove_M1 AND bMotorOn_M1 THEN
    rSetpointTarget_M1 := rSetpointTarget_MinM1;
ELSE
    rSetpointTarget_M1 := rSetpointTarget_MaxM1;
END_IF

// Simulator Reverziranje Motor2 kad uđe u poziciju 
Tgen2(IN:=bInDeadband_M2 , PT:=T#2S , Q=> , ET=> );
R_Tgen2(CLK:=Tgen2.Q , Q=>bTick2 );
IF bTick2 THEN
	bTakt2:=NOT bTakt2;
END_IF

// reverziranje pozicije M2
IF bTakt2 AND bMove_M2 AND bMotorOn_M2  THEN
    rSetpointTarget_M2 := rSetpointTarget_MinM2;
ELSE
    rSetpointTarget_M2 := rSetpointTarget_MaxM2;
END_IF


// MOTOR 1 ===========================
FB_DC_MOTOR1(
	bMotorOn:=bMotorOn_M1,	// Motor ON
	rSetpointTarget:=PRG_ZF_Control.iTargetGear , // Setpopoint Targer pos percent
	rRampRate:=50.0 , // Ramp rate %
	rDeadband:=1.0 , // Deadband pozicije %	 
	rMaxVelocity:=rMaxVelocityM1,	// Zadana brzina %
	rMinVelocity:=10.0,		// Min. brzina %
	cPotMin:= 0.768,             //  V min - krajnji neg. pos.
	cPotMax:= 9.266,             //  V max - krajnji poz. pos.
	rHodMax:= 81.0,             //  max hod spindle mm
	rKp:=rKp_M1 ,	// Kp regulator 5.0
	rLinearPosition_LimMin:= 5.0,	// Safe limit iskljucenja negativan mm 
	rLinearPosition_LimMAx:= 75.0,	// Safe limit iskljucenja pozitivan mm
	rRadno_Min_Pos:= 10.0,	// Radni limit negativan mm
	rRadno_Max_Pos:= 70.0,	// Radni limit pozitivan mm
	rTcy_s:= 0.01, // PLC Tcy u sec
	bHMI_RESET:=bHMI_RESET_M1 , // Reset iz HMI
	iwFeedback:=iwPotFeedback_M1 , // AT %I* Pot feedback Link 
	iwMotorVoltage:=nMotorVoltage_M1 , // AT %I*
	iwMotorCurrent:= nMotorCurrent_M1,  // AT %I*
	ixError:= bError_M1,  // AT %I*
	qwVelocitySetpoint=>nVelocitySetpoint_M1 , // AT %Q*
	qxEnable=>bEnable_M1 , // AT %Q* START MOTORA
	qxReduceTorque=>bReduceTorque_M1 ,// AT %Q* 
	qxReset=>bReset_M1 , // AT %Q*
	rError=>rErrorM1 , // Greska slijedenja pozicije
	bInDeadband=>bInDeadband_M1 , // unutar pozicije
	bSetVelOverPoz=>bSetVelOverPozM1 , // greska set pos koji premasuje INT  - iskljucije Motor
	bSetVelOverNeg=>bSetVelOverNegM1 ,	// greska set pos koji premasuje INT  - iskljucije Motor
	rPotFeedback_Radno_Perc=>rPotFeedback_Radno_PercM1 , //Pozicija % radnog pomaka 0--100%
	rMotorVoltage=>rMotorVoltageM1,	// monitoring napon motora V
	rMotorCurrent=>rMotorCurrentM1 ,		// monitoring struja motora A	
	rActualVelocityRPM=>rActualVelocityRPM_M1,	// trnutna brzina motora RPM
	bErrorLimitPosMin=>bErrorLimitPosMin_M1, // Pozicija ispod min limita 
	bErrorLimitPosMax=>bErrorLimitPosMax_M1,	// Pozicija iznad max limita
	bError=>bERROR_COM_M1,	// generalna greska
	bErrorPos=>bERROR_POS_M1 // greska pozicije ako je van pozicije > 5sec 
);

// MOTOR 2 ===========================
FB_DC_MOTOR2(
	bMotorOn:=bMotorOn_M2,	// Motor ON
	rSetpointTarget:=PRG_ZF_Control.iTargetGas , // Setpopoint Targer pos percent
	rRampRate:=50.0 , // Ramp rate %
	rDeadband:=1.0 , // Deadband pozicije %	 
	rMaxVelocity:=rMaxVelocityM2,	// Zadana brzina %
	rMinVelocity:=10.0,		// Min. brzina %
	cPotMin:= 0.768,             //  V min - krajnji neg. pos.
	cPotMax:= 9.266,             //  V max - krajnji poz. pos.
	rHodMax:= 81.0,             //  max hod spindle mm
	rKp:=rKp_M2 ,	// Kp regulator 5.0
	rLinearPosition_LimMin:= 5.0,	// Safe limit iskljucenja negativan mm 
	rLinearPosition_LimMAx:= 75.0,	// Safe limit iskljucenja pozitivan mm
	rRadno_Min_Pos:= 10.0,	// Radni limit negativan mm
	rRadno_Max_Pos:= 70.0,	// Radni limit pozitivan mm
	rTcy_s:= 0.01, // PLC Tcy u sec
	bHMI_RESET:=bHMI_RESET_M2 , // Reset iz HMI
	iwFeedback:=iwPotFeedback_M2 , // AT %I* Pot feedback Link 
	iwMotorVoltage:=nMotorVoltage_M2 , // AT %I*
	iwMotorCurrent:= nMotorCurrent_M2,  // AT %I*
	ixError:= bError_M2,  // AT %I*
	qwVelocitySetpoint=>nVelocitySetpoint_M2 , // AT %Q*
	qxEnable=>bEnable_M2 , // AT %Q* START MOTORA
	qxReduceTorque=>bReduceTorque_M2 ,// AT %Q* 
	qxReset=>bReset_M2 , // AT %Q*
	rError=>rErrorM2 , // Greska slijedenja pozicije
	bInDeadband=>bInDeadband_M2 , // unutar pozicije
	bSetVelOverPoz=>bSetVelOverPozM2 , // greska set pos koji premasuje INT  - iskljucije Motor
	bSetVelOverNeg=>bSetVelOverNegM2 ,	// greska set pos koji premasuje INT  - iskljucije Motor
	rPotFeedback_Radno_Perc=>rPotFeedback_Radno_PercM2 , //Pozicija % radnog pomaka 0--100%
	rMotorVoltage=>rMotorVoltageM2,	// monitoring napon motora V
	rMotorCurrent=>rMotorCurrentM2 ,		// monitoring struja motora A	
	rActualVelocityRPM=>rActualVelocityRPM_M2,	// trnutna brzina motora RPM
	bErrorLimitPosMin=>bErrorLimitPosMin_M2, // Pozicija ispod min limita 
	bErrorLimitPosMax=>bErrorLimitPosMax_M2,	// Pozicija iznad max limita
	bError=>bERROR_COM_M2,	// generalna greska
	bErrorPos=>bERROR_POS_M2 // greska pozicije ako je van pozicije > 5sec 

);

END_PROGRAM

// ---- POUs/FBs/MeasureRPM.TcPOU
FUNCTION_BLOCK MeasureRPM
VAR_INPUT
	    nPotValue: INT;                    // GVL.iwPotFeedback
END_VAR
VAR_OUTPUT
	nPotValueCount: INT;               
	RPM: LREAL;
	nPotValueGetriba10:DINT; 	// pozicija sim. geriba x10
END_VAR
VAR
	tonPeriodTimer: TON;
	bTick: BOOL;
	nPotValue_Old:INT;
	bRPM: BOOL;
	R_bRPM: R_TRIG;
	RPMcount: INT;
	nPotValueCount10: INT;          //      

	nbRPM: INT;
	bnPotValue: BOOL;
END_VAR

// tonPeriodTimer
tonPeriodTimer(IN:=NOT bTick , PT:=T#10S , Q=>bTick , ET=> );


// na promjenu nPotValue
bnPotValue:=FALSE;
IF (nPotValue <> nPotValue_Old) THEN
	bnPotValue:=TRUE;
END_IF
nPotValue_Old:=	nPotValue;



// Brojanje okretaja + detekcija pada u nulu
bRPM:=FALSE;
IF nPotValue < (nPotValue_Old-(nPotValue-nPotValue_Old)*4) THEN // histereza 20 radi mjerenja u mirovanju
	bRPM:=TRUE;
END_IF

// Brojanje okretaja - detekcija porasta u max
(*
IF nPotValue > (nPotValue_Old+(nPotValue-nPotValue_Old)*4) THEN // histereza 20 radi mjerenja u mirovanju
	bRPM:=TRUE;
END_IF
*)

R_bRPM(CLK:=bRPM , Q=> );
IF R_bRPM.Q THEN
	nPotValueCount:=nPotValueCount+1;	// za RMM
	nPotValueCount10:=nPotValueCount10+1;	// za getribu x 10
	nbRPM:=nbRPM+1;
END_IF

// izracun RPM svake 1Min
IF bTick THEN
	RPMcount:=nPotValueCount;
	RPM:=INT_TO_LREAL(RPMcount*6);
	nPotValueCount:=0;
END_IF

// Simulacija getribe prijenosa 1:10
// broji 10 bRPM

IF (nPotValue > nPotValue_old) AND NOT bRPM THEN
	nPotValueGetriba10:=nPotValueGetriba10 + (nPotValue - nPotValue_old);
END_IF

IF (nPotValue < nPotValue_old) AND NOT bRPM THEN
	nPotValueGetriba10:=nPotValueGetriba10 - (nPotValue_old - nPotValue);
END_IF



// nPotValueGetriba10:=nPotValue + nPotValue*nPotValueCount10;

(*
IF nbRPM>9 THEN
	nbRPM:=0;
	nPotValueCount10:=0;
END_IF
*)

END_FUNCTION_BLOCK

// ---- POUs/FBs/FB_DC_Motor_Direct_Ctrl.TcPOU
FUNCTION_BLOCK FB_DC_Motor_Direct_Ctrl
VAR_INPUT
	bMotorOn: BOOL;			// komanda Motor ON
 	rSetpointTarget: REAL := 50.0;    // Ciljna pozicija % ranga između Min Max
   	rRampRate: REAL := 50.0;          // Brzina rampe [%/s]
    rDeadband: REAL := 2.0;        // Deadband ±%
 	rMaxVelocity: LREAL:= 100.0;
	rMinVelocity: LREAL:= 10.0;
    cPotMin: REAL := 0.768;             //  V min - krajnji neg. pos.
    cPotMax: REAL := 9.266;             //  V max - krajnji poz. pos.
	rHodMax: REAL := 81.0;             //  max hod spindle mm
	rKp: REAL := 10;              // P pojačanje
 	rLinearPosition_LimMin: REAL:= 5.0;	// Safe limit iskljucenja negativan mm
	rLinearPosition_LimMAx: REAL:= 75.0;	// Safe limit iskljucenja pozitivan mm
 	rRadno_Min_Pos: REAL:= 10.0;	// Radni limit negativan mm
	rRadno_Max_Pos: REAL:= 70.0;	// Radni limit pozitivan mm

	rTcy_s: REAL:=0.01;	// PLC Tcy u sec
  	// Realni Potenciometar - u RAW vrijednosti napona
	bHMI_RESET: BOOL;	// Reset iz HMI
	
	iwFeedback: INT;	// AT %I* Pot feedback Link 
	iwMotorVoltage : UINT; // AT %I* Info data 1 (mV)
	iwMotorCurrent : UINT; // AT %I* Info data 2 (mA)
	ixError : BOOL; // AT %I* Error

END_VAR
VAR_OUTPUT
    qwVelocitySetpoint : INT; // AT %Q* Link na "Velocity" (49.0)
	qxEnable : BOOL;         // AT %Q* DCM Control Channel 1.Enable
	qxReduceTorque : BOOL;   // AT %Q* DCM Control Channel 1.Reduce torque
	qxReset : BOOL;          // AT %Q* DCM Control Channel 1.Reset  

	rError: REAL;	// greska slijeđenja
	bInDeadband: BOOL;	// unutar pozicije
	bSetVelOverPoz: BOOL;	// setpoint koji premasuje INT 
	bSetVelOverNeg: BOOL;	// setpoint koji premasuje INT 
	rPotFeedback_Radno_Perc: LREAL;	//Postotak radnog pomaka 0--100% mora biti unutar Safe limita
	rMotorVoltage: REAL;	// monitoring V
	rMotorCurrent: REAL;	// monitoring A
	rActualVelocityRPM: REAL;	// Stvarna brzina [RPM]
	bErrorLimitPosMin: BOOL;	// Pozicija ispod min limita 
	bErrorLimitPosMax: BOOL;	// Pozicija iznad max limita 
	bError: BOOL;	// Generalna greska  
	bErrorPos: BOOL;	// greska pozicije ako je van pozicije > n sec  
	
END_VAR
VAR
	rSetpoint: REAL ;      // Željena pozicija 0-100%
	rPotFeedback_V: REAL;		// Feedback napon
	rLinearPosition: REAL;		// stvarna pozicija mm 

	Kn: LREAL;	// faktor napona motora 320
	
	rVelocitySetpoint: LREAL;	// velocity setpoint
	rVelocityCmd: LREAL;
	fbVelocityTimer: TON;	// Timer za uzorkovanje
    tSampleTime: TIME := T#50MS;  // Vrijeme uzorkovanja
	rDeltaPosition: LREAL;	// Promjena pozicije
	rLastPosition: REAL;	// Prethodna pozicija
	rActualVelocity: LREAL;	// Stvarna brzina [%/s]
	rVelocityFiltered: LREAL; // Stvarna brzina [%/s] filter
	rFilterConst: REAL := 0.3;    // Filter konstanta (0.1-0.5)
	bMotorOnCmd: BOOL;
	TON_bInDeadband: TON;
END_VAR

// FB za DC Motor

// Rampiranje setpointa
IF rSetpoint < rSetpointTarget - 0.1 THEN
    // Rampiranje gore
    rSetpoint := rSetpoint + rRampRate * rTcy_s; // 0.01 = 10ms ciklus
    IF rSetpoint > rSetpointTarget THEN
        rSetpoint := rSetpointTarget;
    END_IF
ELSIF rSetpoint > rSetpointTarget + 0.1 THEN
    // Rampiranje dolje  
    rSetpoint := rSetpoint - rRampRate * rTcy_s;
    IF rSetpoint < rSetpointTarget THEN
        rSetpoint := rSetpointTarget;
    END_IF
END_IF

// Skaliranje 1 okretajng pot pozicije - EL3255.
rPotFeedback_V:=10.0*iwFeedback/32767;	//napon na ulazu u EL3255
// pozicija pomaka = 81mm
rLinearPosition:=rHodMax*(rPotFeedback_V-cPotMin)/(cPotMax-cPotMin);

// Sigurnosni limiti + / - hoda 0-->     <--rHodMax   - iskljucuju Motor
bErrorLimitPosMin:=FALSE;	
bErrorLimitPosMax:=FALSE;	
IF (rLinearPosition < rLinearPosition_LimMin) THEN
	bErrorLimitPosMin:=TRUE;	
END_IF
IF (rLinearPosition > rLinearPosition_LimMAx) THEN
	bErrorLimitPosMax:=TRUE;	
END_IF

IF bErrorLimitPosMin OR bErrorLimitPosMax THEN
	bMotorOnCmd:=FALSE;
ELSE
	bMotorOnCmd:=bMotorOn;	
END_IF

// Radno podrucje pomaka 0..100% = MORA BITI UNUTAR SIGURNOSNIH LIMITA
rPotFeedback_Radno_Perc:= 100*(rLinearPosition-rRadno_Min_Pos)/(rRadno_Max_Pos-rRadno_Min_Pos);

// Open-loop kontrola
// Setpoint 0..100% = 0.....
// Limit za pretvorbu u integer 
// greska ako je veće od 32766 i manje od - 32766

// Kn ke multiplikator za setpoint u granicama -32000 .. 32000 / 0.100%
Kn:=320; // ako ide do napona napajanja 12V onda na 100% steka
// reset iz HMI
// bReset := FALSE;
IF bHMI_RESET THEN
	bSetVelOverPoz:=FALSE;
	bSetVelOverNeg:=FALSE;
    qxReset := TRUE;
END_IF

IF NOT ixError THEN
	qxReset := FALSE;
END_IF

// greška / iskljucenje motora ako bi setpoint prešao INT max - da ne okrene u drigi smjer !
IF (rVelocitySetpoint*Kn > 32766) THEN
	bSetVelOverPoz:=TRUE;
END_IF
IF (rVelocitySetpoint*Kn < -32766) THEN
	bSetVelOverNeg:=TRUE;
END_IF
IF bSetVelOverPoz OR bSetVelOverNeg THEN
	bMotorOnCmd:=FALSE;
ELSE
	// ako je ispravan setpoint brzine - računa INT z aizlaz
	qwVelocitySetpoint:=LREAL_TO_INT(rVelocitySetpoint*Kn);
END_IF

// POZICIJSKA REGULACIJA
    // Računaj grešku pozicije
    rError := rSetpoint - rPotFeedback_Radno_Perc;
    
    // Provjeri deadband
    bInDeadband := ABS(rError) <= rDeadband;
	// Greska pozicije ako je izvan rDeadband > n sec
TON_bInDeadband(IN:=NOT bInDeadband , PT:=T#5S , Q=>bErrorPos , ET=> );
	
IF bMotorOn THEN
    
    IF NOT bInDeadband THEN
        // P regulator
        rVelocityCmd := rError * rKp;
        
        // Ograniči na max brzinu
        rVelocityCmd := LIMIT(-rMaxVelocity, rVelocityCmd, rMaxVelocity);
        
        // Primjeni minimalnu brzinu
        IF (ABS(rVelocityCmd) > 0.1) AND (ABS(rVelocityCmd) < rMinVelocity) THEN
            IF rVelocityCmd > 0 THEN
                rVelocityCmd := rMinVelocity;
            ELSE
                rVelocityCmd := -rMinVelocity;
            END_IF
        END_IF
    ELSE
        // Unutar deadband - zaustavi
        rVelocityCmd := 0.0;
    END_IF
    
    // Postavi brzinu
    rVelocitySetpoint := rVelocityCmd;
ELSE
    rVelocitySetpoint := 0.0;
END_IF

// Računanje brzine iz promjene pozicije

// Timer za periodičko računanje brzine
fbVelocityTimer(IN:= NOT fbVelocityTimer.Q, PT:= tSampleTime);

// Računaj brzinu kada timer istekne
IF fbVelocityTimer.Q THEN
    // Promjena pozicije u %
    rDeltaPosition := rLinearPosition - rLastPosition;
    
    // Brzina u mm/s !!!! NAVOJ IMA MULTIPLIKATOR X2
    rActualVelocity := rDeltaPosition / 0.05 / 2 ; // 50ms = 0.05s
    
    // Spremi trenutnu poziciju
    rLastPosition := rLinearPosition;
    
    // Filter brzine (PT1)
    rVelocityFiltered := rVelocityFiltered * (1.0 - rFilterConst) + 
                        rActualVelocity * rFilterConst;
END_IF

// Preračun u druge jedinice
// 81mm =  171.3 okr Motora
// RPM motora
rActualVelocityRPM := 60*171.3*rActualVelocity/81 ;


// =======================  DIVER PREMA TERMINALU

// driver prema EL7342
IF bMotorOnCmd THEN
    qxEnable := TRUE;
    qxReduceTorque := FALSE;  // Puna snaga
 ELSE
    qxEnable := FALSE;
    qxReduceTorque := FALSE;
    qwVelocitySetpoint := 0;
END_IF

// Monitoring Napona - struje motora
rMotorVoltage:=(UINT_TO_INT(iwMotorVoltage))/1000.0;
rMotorCurrent:=(UINT_TO_INT(iwMotorCurrent))/1000.0;

// Generalna greska, terminal, set pos, Limit feedback
bError:=ixError OR 
bSetVelOverPoz OR 
bSetVelOverNeg OR 
bErrorLimitPosMin OR 
bErrorLimitPosMax OR
bErrorPos;

END_FUNCTION_BLOCK

// ---- POUs/PRG_Engine.TcPOU
PROGRAM PRG_Engine
VAR
    (* Instanca glavnog bloka za kontrolu motora (Prošireni s prethodnim uputama) *)
    fbEngine        : FB_EngineControl;
    fbStation       : FB_StationManager;

    (* Triggeri za tipke ID10 i ID11 *)
    rtMode_ID10     : R_TRIG;
    rtMode_ID11     : R_TRIG;
    iModeState      : INT; (* 0=OFF, 1=Propulsion (Green), 2=Ballast Ready (Blue) *)

    (* Interne varijable za logiku *)
    bInterlockDoors : BOOL;
    bValvePathReady : BOOL; (* Barem jedan ventil otvoren *)
    bInterlockTotal : BOOL; (* Konačna dozvola za turbinu *)
    bBallastActive  : BOOL; (* Zastavica: Balasti rade *)
    bWinchReq       : BOOL; (* Zastavica: Netko želi koristiti vinč *)
	
	(* Triggeri za tipke *)
    rtStart_ID10, rtStart_ID11 : R_TRIG;
    rtStop_ID10,  rtStop_ID11  : R_TRIG;
    rtSel_ID10,   rtSel_ID11   : R_TRIG;

    (* Timeri za Start sekvencu *)
    tonStartDelay   : TON;   (* Kašnjenje startera nakon Ignitiona *)
    toffStartHold   : TOF;  (* Drži starter aktivnim kratko nakon puštanja tipke *)
    
    (* Timeri za Stop sekvencu *)
    tmrStopSequence : TON;
    
    (* Interne statusne varijable *)
    bIgnitionActive : BOOL; 
    bEngineRunning  : BOOL;
    bStartButtonPressed : BOOL; (* Pomoćna varijabla za detekciju pritiska *)
    iActiveStation  : INT := 1;
END_VAR

(* ========================================================= *)
(* 1. STATION MANAGER & VIZUALIZACIJA (Tipka 3)              *)
(* ========================================================= *)
fbStation(
    bBtn1 := GVL_CAN.ID10_Status[3], 
    bBtn2 := GVL_CAN.ID11_Status[3],
    iPot1 := GVL_IO.iLever_St1_Raw,
    iPot2 := GVL_IO.iLever_St2_Raw,
    bActiveSt1 => GVL_IO.bLed_Sel_St1,
    bActiveSt2 => GVL_IO.bLed_Sel_St2,
    bBuzzerOut => GVL_IO.bBuzzer,
    iSelectedPot => GVL_IO.iActiveLever_Raw
);

// --- 1. STATUS MOTORA ---
bEngineRunning := bIgnitionActive OR (GVL_IO.fEngineRPM_Scaled > 400.0);
bStartButtonPressed := GVL_CAN.ID10_Status[1] OR GVL_CAN.ID11_Status[1];

// --- 2. LOGIKA STARTA (Tipka 1) ---
rtStart_ID10(CLK := GVL_CAN.ID10_Status[1]);
rtStart_ID11(CLK := GVL_CAN.ID11_Status[1]);

// A) Setiranje Ignitiona na prvi klik
IF (rtStart_ID10.Q OR rtStart_ID11.Q) AND NOT bIgnitionActive THEN
    bIgnitionActive := TRUE;
END_IF

// B) TON: Čekaj npr. 500ms nakon što je Ignition aktivan prije nego dozvoliš Start
tonStartDelay(IN := bStartButtonPressed AND bIgnitionActive AND NOT bEngineRunning, 
              PT := T#500MS);

// C) TOFF: Drži DO_Start aktivnim npr. 200ms nakon puštanja tipke (da izbjegnemo "ckatanje" releja)
toffStartHold(IN := tonStartDelay.Q, 
              PT := T#200MS);

// Fizički izlaz za Starter
GVL_IO.DO_Engine_Starter := toffStartHold.Q;

// --- 3. LOGIKA STOPA (Tipka 2) ---
rtStop_ID10(CLK := GVL_CAN.ID10_Status[2]);
rtStop_ID11(CLK := GVL_CAN.ID11_Status[2]);

IF (rtStop_ID10.Q OR rtStop_ID11.Q) AND bIgnitionActive THEN
    GVL_IO.DO_Engine_Stop := TRUE;
END_IF

tmrStopSequence(IN := GVL_IO.DO_Engine_Stop, PT := T#2S);

IF tmrStopSequence.Q THEN
    GVL_IO.DO_Engine_Stop := FALSE;
    bIgnitionActive := FALSE;
END_IF

// --- 4. ODABIR KOMANDE (Tipka 3) ---
rtSel_ID10(CLK := GVL_CAN.ID10_Status[3]);
rtSel_ID11(CLK := GVL_CAN.ID11_Status[3]);
IF rtSel_ID10.Q THEN iActiveStation := 1; END_IF
IF rtSel_ID11.Q THEN iActiveStation := 2; END_IF

// --- 5. VIZUALIZACIJA (Boje na tipkovnicama) ---

// TIPKA 1 (START)
IF bStartButtonPressed THEN
    GVL_CAN.ID10_Config[1].Boja := GVL_CAN.ID11_Config[1].Boja := 2; // ZELENO (Radi)
    GVL_CAN.ID10_Config[1].Blink := GVL_CAN.ID11_Config[1].Blink := TRUE;
ELSIF bEngineRunning  THEN
    GVL_CAN.ID10_Config[1].Boja := GVL_CAN.ID11_Config[1].Boja := 2; // Zeleno (Vergla)
    GVL_CAN.ID10_Config[1].Blink := GVL_CAN.ID11_Config[1].Blink := FALSE;                           // Blinka 
ELSE
    GVL_CAN.ID10_Config[1].Boja := GVL_CAN.ID11_Config[1].Boja := 0; // OFF
    GVL_CAN.ID10_Config[1].Blink := FALSE;
END_IF

// TIPKA 2 (STOP)
IF GVL_IO.DO_Engine_Stop THEN
    GVL_CAN.ID10_Config[2].Boja := GVL_CAN.ID11_Config[2].Boja := 1; 
    GVL_CAN.ID10_Config[2].Blink := GVL_CAN.ID11_Config[2].Blink := TRUE; // Blinka crveno dok traje stop sekvenca
ELSIF bIgnitionActive THEN
    GVL_CAN.ID10_Config[2].Boja := GVL_CAN.ID11_Config[2].Boja := 1; 
    GVL_CAN.ID10_Config[2].Blink := GVL_CAN.ID11_Config[2].Blink := FALSE;
ELSE
    GVL_CAN.ID10_Config[2].Boja := GVL_CAN.ID11_Config[2].Boja := 0;
END_IF

// TIPKA 3 (SEL)
IF iActiveStation = 1 THEN
    GVL_CAN.ID10_Config[3].Boja := 4; GVL_CAN.ID11_Config[3].Boja := 0;
ELSE
    GVL_CAN.ID10_Config[3].Boja := 0; GVL_CAN.ID11_Config[3].Boja := 4;
END_IF

// --- 6. FIZIČKI IZLAZ KONTAKTA ---
GVL_IO.DO_Engine_Ignition := bIgnitionActive;

END_PROGRAM

// ---- POUs/FBs/FB_EngineControl.TcPOU
FUNCTION_BLOCK FB_EngineControl
VAR_INPUT
    (* Kontrola rada motora (Novi zahtjevi) *)
    bBtnStart      : BOOL;          (* Tipka 1 - Start *)
    bBtnStop       : BOOL;          (* Tipka 2 - Stop *)
    bModeProp      : BOOL;          (* Tipka 4 - Mode (Zelena) *)
    bModeBallast   : BOOL;          (* Tipka 4 - Mode (Plava) *)

    (* Postojeći ulazi tvojeg FB-a *)
    fRpmCurrent    : REAL;          (* Trenutni RPM motora *)
    fThrottleIn    : REAL;          (* Ručica gasa (0-100%) *)
    eGearIn        : INT;           (* Željena brzina (Joystick: 0=N, 1=FWD, 2=REV) *)
    bDoorsOk       : BOOL;          (* Interlock: Vrata otvorena *)
    fRpmLimit      : REAL := 900.0; (* Max RPM za šaltanje *)
    tNeutralDelay  : TIME := T#1500MS; 
END_VAR

VAR_OUTPUT
    (* Izlazi prema hardveru *)
    bIgnition      : BOOL;          (* Relej kontakta *)
    bStarter       : BOOL;          (* Relej elektropokretača *)
    fThrottleOut   : REAL;          (* Izlaz prema motoru *)
    eGearOut       : INT;           (* Izlaz prema kopči (0=N, 1=FWD, 2=REV) *)

    (* Statusi za vizualizaciju tipki *)
    iColorStart    : INT;           (* Boja za Tipku 1 *)
    iColorStop     : INT;           (* Boja za Tipku 2 *)
    bEngineRunning : BOOL;          (* Status: Motor radi *)
    bShifting      : BOOL;          (* Status: Mijenjanje brzine *)
    bHighRpmLock   : BOOL;          (* Status: Zabrana šaltanja *)
END_VAR

VAR
    (* Interni tajmeri i varijable *)
    rtStart        : R_TRIG;
    tmrRunDelay    : TON;           (* Simulacija feedbacka motora *)
    stepShift      : INT := 0;      (* State machine šaltanja *)
    tmrDelay       : TON;           (* Timer za sekvencu šaltanja *)
    eTargetGear    : INT;           
END_VAR


// ===========================================================
// 1. LOGIKA START / STOP I IGNITION
// ===========================================================
rtStart(CLK := bBtnStart);

// START: Ako stisnem start, pali Ignition. Starter vrti dok držim tipku.
IF rtStart.Q AND NOT bEngineRunning THEN
    bIgnition := TRUE;
END_IF

// Starter radi samo ako imamo Ignition, držimo tipku i motor još ne radi
bStarter := bBtnStart AND bIgnition AND NOT bEngineRunning;

// Simulacija da je motor upalio (feedback) - zeleno svjetlo nakon 2s startera
tmrRunDelay(IN := bStarter, PT := T#2S);
IF tmrRunDelay.Q THEN
    bEngineRunning := TRUE;
END_IF

// STOP: Gasi motor i RESETIRA Ignition (kako si tražio)
// Ako fali ignition, stop ne radi (uvjet bIgnition)
IF bBtnStop AND bIgnition THEN
    bIgnition := FALSE;
    bEngineRunning := FALSE;
END_IF

// Reset Ignitiona ako motor nekako stane (opcionalno sigurnosno)
IF NOT bEngineRunning AND NOT bStarter AND bIgnition AND bBtnStop THEN
     bIgnition := FALSE;
END_IF

// ===========================================================
// 2. LOGIKA ŠALTANJA (Tvoj postojeći State Machine)
// ===========================================================

// Interlock: Ako su vrata zatvorena ILI nismo u Propulsion modu -> NEUTRAL
// Dodajemo uvjet bModeProp: Kopča radi samo ako je Mode Zeleni
IF NOT bDoorsOk OR NOT bModeProp THEN
    eTargetGear := 0; 
ELSE
    eTargetGear := eGearIn;
END_IF

CASE stepShift OF
    0: // STABILNO STANJE
        // Gas ide van samo ako motor radi i ne šaltamo
        IF bEngineRunning AND NOT bShifting THEN
            fThrottleOut := fThrottleIn;
        ELSE
            fThrottleOut := 0.0;
        END_IF

        // Provjera promjene brzine
        IF eTargetGear <> eGearOut AND bEngineRunning THEN
            IF fRpmCurrent > fRpmLimit THEN
                bHighRpmLock := TRUE;
                fThrottleOut := 0.0; 
            ELSE
                bHighRpmLock := FALSE;
                bShifting := TRUE;
                stepShift := 10;
            END_IF
        ELSE
            bHighRpmLock := FALSE;
        END_IF

    10: // PRIPREMA - SPUSTI GAS
        fThrottleOut := 0.0; 
        tmrDelay(IN := TRUE, PT := T#200MS);
        IF tmrDelay.Q THEN tmrDelay(IN := FALSE); stepShift := 20; END_IF

    20: // IZBACI U NEUTRAL
        eGearOut := 0;
        IF eTargetGear = 0 THEN stepShift := 99; ELSE stepShift := 30; END_IF

    30: // PAUZA U NEUTRALU
        tmrDelay(IN := TRUE, PT := tNeutralDelay);
        IF tmrDelay.Q THEN tmrDelay(IN := FALSE); stepShift := 40; END_IF

    40: // UBACI U BRZINU
        eGearOut := eTargetGear;
        tmrDelay(IN := TRUE, PT := T#500MS);
        IF tmrDelay.Q THEN tmrDelay(IN := FALSE); stepShift := 99; END_IF

    99: // KRAJ SEKVENCE
        bShifting := FALSE;
        stepShift := 0;
END_CASE

// ===========================================================
// 3. VIZUALIZACIJA BOJA (Za tipkovnice)
// ===========================================================

// Tipka 1 (Start): Plava kad je kontakt, Zelena kad motor radi
IF bEngineRunning THEN
    iColorStart := 2; // Green
ELSIF bIgnition THEN
    iColorStart := 4; // Blue
ELSE
    iColorStart := 0; // Off
END_IF

// Tipka 2 (Stop): Crvena ako je kontakt uključen
IF bIgnition THEN
    iColorStop := 1; // Red
ELSE
    iColorStop := 0; // Off
END_IF

END_FUNCTION_BLOCK

// ---- POUs/FBs/FB_StationManager.TcPOU
FUNCTION_BLOCK FB_StationManager
VAR_INPUT
    (* Ulazi s ručica *)
    bBtn1, bBtn2      : BOOL;
    iPot1, iPot2      : INT;
    
    (* Kalibracija Neutrala *)
    iNeutCenter       : INT := 16000; (* Sredina *)
    iNeutTol          : INT := 2000;  (* Tolerancija +/- *)
END_VAR

VAR_OUTPUT
    (* Tko je aktivan? *)
    bActiveSt1        : BOOL;
    bActiveSt2        : BOOL;
    
    (* Signal za buzzer *)
    bBuzzerOut        : BOOL;
    
    (* Odabrani potenciometar *)
    iSelectedPot      : INT;
END_VAR

VAR
    (* Interno *)
    bRequest1, bRequest2 : BOOL; (* Detekcija pritiska (Rising Edge) *)
    rtBtn1, rtBtn2       : R_TRIG; (* Triggeri za tipke *)
    
    bSafeToTransfer      : BOOL;
    tmrBuzzer            : TP;     (* Timer za Bip-Bip *)
    iBipCount            : INT;    (* Brojač bipova *)
    fbPulse              : TON;    (* Za blinkanje buzzera *)
END_VAR

// --- KOD ---

// 1. Detekcija pritiska tipke
rtBtn1(CLK := bBtn1);
rtBtn2(CLK := bBtn2);

// 2. Provjera jesu li ručice u Neutralu?
// Obje moraju biti blizu sredine da bi transfer bio siguran
bSafeToTransfer := (ABS(iPot1 - iNeutCenter) < iNeutTol) AND 
                   (ABS(iPot2 - iNeutCenter) < iNeutTol);

// 3. Logika prebacivanja (Transfer)

// A) Zahtjev za Stanicu 1
IF rtBtn1.Q THEN
    IF bSafeToTransfer THEN
        bActiveSt1 := TRUE;
        bActiveSt2 := FALSE;
    ELSE
        // Nije sigurno! Pali alarm
        iBipCount := 3; // 3 puta bipni
    END_IF
END_IF

// B) Zahtjev za Stanicu 2
IF rtBtn2.Q THEN
    IF bSafeToTransfer THEN
        bActiveSt1 := FALSE;
        bActiveSt2 := TRUE;
    ELSE
        // Nije sigurno! Pali alarm
        iBipCount := 3;
    END_IF
END_IF

// Defaultno stanje na paljenju (npr. Stanica 1)
IF NOT bActiveSt1 AND NOT bActiveSt2 THEN
    bActiveSt1 := TRUE;
END_IF


// 4. Odabir signala
IF bActiveSt1 THEN
    iSelectedPot := iPot1;
ELSE
    iSelectedPot := iPot2;
END_IF


// 5. Logika Buzzera 
IF iBipCount > 0 THEN
    // Generiraj puls (npr. 200ms ON, 200ms OFF)
    fbPulse(IN := NOT fbPulse.Q, PT := T#200MS);
    
    IF fbPulse.Q THEN
        // Svaki drugi puls smanji brojač (da dobijemo ON-OFF ciklus)
        // (Ovo je pojednostavljeno, može se i ljepše s CASE-om)
    END_IF
    
    // Buzzer prati puls
    bBuzzerOut := fbPulse.ET < T#100MS; // Prvih 100ms sviraj
    
    // Odbrojavanje (Ovo je pseudo-kod, u stvarnosti trebaš state machine za biper)
    // Ali za jednostavnost: Neka svira dok je tipka stisnuta ako nije Safe?
    // Ili jednostavnije:
    
    // --- JEDNOSTAVNIJI ALARM ---
    // Ako stisneš tipku a nije safe -> Buzzer radi dok držiš tipku
    if (bBtn1 OR bBtn2) AND NOT bSafeToTransfer THEN
        bBuzzerOut := TRUE;
    ELSE
        bBuzzerOut := FALSE;
    END_IF
END_IF

END_FUNCTION_BLOCK

// ---- POUs/PRG_BlinkMarine.TcPOU
PROGRAM PRG_BlinkMarine
VAR
    i : INT;
    BitMask : DWORD; // Pomoćna varijabla za rad s bitovima
END_VAR


// ==========================================
// OBRADA ID10 (4 tipke - USINT)
// ==========================================
GVL_CAN.ID10_LedRed := 0; GVL_CAN.ID10_LedGreen := 0; GVL_CAN.ID10_LedBlue := 0;
GVL_CAN.ID10_LedBlinkRed := 0; GVL_CAN.ID10_LedBlinkGreen := 0; GVL_CAN.ID10_LedBlinkBlue := 0;

FOR i := 1 TO 4 DO
    BitMask := SHL(DWORD#1, i-1);
    
    // Čitanje statusa tipke
    GVL_CAN.ID10_Status[i] := (GVL_CAN.ID10_KeyState AND DWORD_TO_USINT(BitMask)) > 0;
    
    // Logika boja
    // CRVENA (Red, Yellow, Magenta, White, Amber, Orange)
    IF GVL_CAN.ID10_Config[i].Boja = E_BlinkMarine_Color.RED OR 
       GVL_CAN.ID10_Config[i].Boja = E_BlinkMarine_Color.YELLOW OR 
       GVL_CAN.ID10_Config[i].Boja = E_BlinkMarine_Color.MAGENTA OR 
       GVL_CAN.ID10_Config[i].Boja = E_BlinkMarine_Color.WHITE OR
       GVL_CAN.ID10_Config[i].Boja = E_BlinkMarine_Color.AMBER OR
       GVL_CAN.ID10_Config[i].Boja = E_BlinkMarine_Color.ORANGE THEN
        GVL_CAN.ID10_LedRed := GVL_CAN.ID10_LedRed OR DWORD_TO_USINT(BitMask);
    END_IF
    
    // ZELENA (Green, Yellow, Cyan, White, Amber, Orange)
    IF GVL_CAN.ID10_Config[i].Boja = E_BlinkMarine_Color.GREEN OR 
       GVL_CAN.ID10_Config[i].Boja = E_BlinkMarine_Color.YELLOW OR 
       GVL_CAN.ID10_Config[i].Boja = E_BlinkMarine_Color.CYAN OR 
       GVL_CAN.ID10_Config[i].Boja = E_BlinkMarine_Color.WHITE OR
       GVL_CAN.ID10_Config[i].Boja = E_BlinkMarine_Color.AMBER OR
       GVL_CAN.ID10_Config[i].Boja = E_BlinkMarine_Color.ORANGE THEN
        GVL_CAN.ID10_LedGreen := GVL_CAN.ID10_LedGreen OR DWORD_TO_USINT(BitMask);
    END_IF
    
    // PLAVA (Blue, Magenta, Cyan, White)
    IF GVL_CAN.ID10_Config[i].Boja = E_BlinkMarine_Color.BLUE OR 
       GVL_CAN.ID10_Config[i].Boja = E_BlinkMarine_Color.MAGENTA OR 
       GVL_CAN.ID10_Config[i].Boja = E_BlinkMarine_Color.CYAN OR 
       GVL_CAN.ID10_Config[i].Boja = E_BlinkMarine_Color.WHITE THEN
        GVL_CAN.ID10_LedBlue := GVL_CAN.ID10_LedBlue OR DWORD_TO_USINT(BitMask);
    END_IF
    
    // BLINK LOGIKA
    IF GVL_CAN.ID10_Config[i].Blink THEN
        IF (GVL_CAN.ID10_LedRed AND DWORD_TO_USINT(BitMask)) > 0 THEN GVL_CAN.ID10_LedBlinkRed := GVL_CAN.ID10_LedBlinkRed OR DWORD_TO_USINT(BitMask); END_IF
        IF (GVL_CAN.ID10_LedGreen AND DWORD_TO_USINT(BitMask)) > 0 THEN GVL_CAN.ID10_LedBlinkGreen := GVL_CAN.ID10_LedBlinkGreen OR DWORD_TO_USINT(BitMask); END_IF
        IF (GVL_CAN.ID10_LedBlue AND DWORD_TO_USINT(BitMask)) > 0 THEN GVL_CAN.ID10_LedBlinkBlue := GVL_CAN.ID10_LedBlinkBlue OR DWORD_TO_USINT(BitMask); END_IF
    END_IF
END_FOR

// ==========================================
// OBRADA ID11 (4 tipke - Kopija logike ID10)
// ==========================================
GVL_CAN.ID11_LedRed := 0; GVL_CAN.ID11_LedGreen := 0; GVL_CAN.ID11_LedBlue := 0;
GVL_CAN.ID11_LedBlinkRed := 0; GVL_CAN.ID11_LedBlinkGreen := 0; GVL_CAN.ID11_LedBlinkBlue := 0;

FOR i := 1 TO 4 DO
    BitMask := SHL(DWORD#1, i-1);
    GVL_CAN.ID11_Status[i] := (GVL_CAN.ID11_KeyState AND DWORD_TO_USINT(BitMask)) > 0;
    
    IF GVL_CAN.ID11_Config[i].Boja = E_BlinkMarine_Color.RED OR GVL_CAN.ID11_Config[i].Boja = E_BlinkMarine_Color.YELLOW OR GVL_CAN.ID11_Config[i].Boja = E_BlinkMarine_Color.MAGENTA OR GVL_CAN.ID11_Config[i].Boja = E_BlinkMarine_Color.WHITE OR GVL_CAN.ID11_Config[i].Boja = E_BlinkMarine_Color.AMBER OR GVL_CAN.ID11_Config[i].Boja = E_BlinkMarine_Color.ORANGE THEN
        GVL_CAN.ID11_LedRed := GVL_CAN.ID11_LedRed OR DWORD_TO_USINT(BitMask);
    END_IF
    IF GVL_CAN.ID11_Config[i].Boja = E_BlinkMarine_Color.GREEN OR GVL_CAN.ID11_Config[i].Boja = E_BlinkMarine_Color.YELLOW OR GVL_CAN.ID11_Config[i].Boja = E_BlinkMarine_Color.CYAN OR GVL_CAN.ID11_Config[i].Boja = E_BlinkMarine_Color.WHITE OR GVL_CAN.ID11_Config[i].Boja = E_BlinkMarine_Color.AMBER OR GVL_CAN.ID11_Config[i].Boja = E_BlinkMarine_Color.ORANGE THEN
        GVL_CAN.ID11_LedGreen := GVL_CAN.ID11_LedGreen OR DWORD_TO_USINT(BitMask);
    END_IF
    IF GVL_CAN.ID11_Config[i].Boja = E_BlinkMarine_Color.BLUE OR GVL_CAN.ID11_Config[i].Boja = E_BlinkMarine_Color.MAGENTA OR GVL_CAN.ID11_Config[i].Boja = E_BlinkMarine_Color.CYAN OR GVL_CAN.ID11_Config[i].Boja = E_BlinkMarine_Color.WHITE THEN
        GVL_CAN.ID11_LedBlue := GVL_CAN.ID11_LedBlue OR DWORD_TO_USINT(BitMask);
    END_IF
    IF GVL_CAN.ID11_Config[i].Blink THEN
        IF (GVL_CAN.ID11_LedRed AND DWORD_TO_USINT(BitMask)) > 0 THEN GVL_CAN.ID11_LedBlinkRed := GVL_CAN.ID11_LedBlinkRed OR DWORD_TO_USINT(BitMask); END_IF
        IF (GVL_CAN.ID11_LedGreen AND DWORD_TO_USINT(BitMask)) > 0 THEN GVL_CAN.ID11_LedBlinkGreen := GVL_CAN.ID11_LedBlinkGreen OR DWORD_TO_USINT(BitMask); END_IF
        IF (GVL_CAN.ID11_LedBlue AND DWORD_TO_USINT(BitMask)) > 0 THEN GVL_CAN.ID11_LedBlinkBlue := GVL_CAN.ID11_LedBlinkBlue OR DWORD_TO_USINT(BitMask); END_IF
    END_IF
END_FOR

// ==========================================
// OBRADA ID20 (15 tipki - UINT)
// ==========================================
GVL_CAN.ID20_LedRed := 0; GVL_CAN.ID20_LedGreen := 0; GVL_CAN.ID20_LedBlue := 0;
GVL_CAN.ID20_LedBlinkRed := 0; GVL_CAN.ID20_LedBlinkGreen := 0; GVL_CAN.ID20_LedBlinkBlue := 0;

FOR i := 1 TO 15 DO
    BitMask := SHL(DWORD#1, i-1);
    
    GVL_CAN.ID20_Status[i] := (GVL_CAN.ID20_KeyState AND DWORD_TO_UINT(BitMask)) > 0;
    
    IF GVL_CAN.ID20_Config[i].Boja = E_BlinkMarine_Color.RED OR GVL_CAN.ID20_Config[i].Boja = E_BlinkMarine_Color.YELLOW OR GVL_CAN.ID20_Config[i].Boja = E_BlinkMarine_Color.MAGENTA OR GVL_CAN.ID20_Config[i].Boja = E_BlinkMarine_Color.WHITE OR GVL_CAN.ID20_Config[i].Boja = E_BlinkMarine_Color.AMBER OR GVL_CAN.ID20_Config[i].Boja = E_BlinkMarine_Color.ORANGE THEN
        GVL_CAN.ID20_LedRed := GVL_CAN.ID20_LedRed OR DWORD_TO_UINT(BitMask);
    END_IF
    IF GVL_CAN.ID20_Config[i].Boja = E_BlinkMarine_Color.GREEN OR GVL_CAN.ID20_Config[i].Boja = E_BlinkMarine_Color.YELLOW OR GVL_CAN.ID20_Config[i].Boja = E_BlinkMarine_Color.CYAN OR GVL_CAN.ID20_Config[i].Boja = E_BlinkMarine_Color.WHITE OR GVL_CAN.ID20_Config[i].Boja = E_BlinkMarine_Color.AMBER OR GVL_CAN.ID20_Config[i].Boja = E_BlinkMarine_Color.ORANGE THEN
        GVL_CAN.ID20_LedGreen := GVL_CAN.ID20_LedGreen OR DWORD_TO_UINT(BitMask);
    END_IF
    IF GVL_CAN.ID20_Config[i].Boja = E_BlinkMarine_Color.BLUE OR GVL_CAN.ID20_Config[i].Boja = E_BlinkMarine_Color.MAGENTA OR GVL_CAN.ID20_Config[i].Boja = E_BlinkMarine_Color.CYAN OR GVL_CAN.ID20_Config[i].Boja = E_BlinkMarine_Color.WHITE THEN
        GVL_CAN.ID20_LedBlue := GVL_CAN.ID20_LedBlue OR DWORD_TO_UINT(BitMask);
    END_IF
    
    IF GVL_CAN.ID20_Config[i].Blink THEN
        IF (GVL_CAN.ID20_LedRed AND DWORD_TO_UINT(BitMask)) > 0 THEN GVL_CAN.ID20_LedBlinkRed := GVL_CAN.ID20_LedBlinkRed OR DWORD_TO_UINT(BitMask); END_IF
        IF (GVL_CAN.ID20_LedGreen AND DWORD_TO_UINT(BitMask)) > 0 THEN GVL_CAN.ID20_LedBlinkGreen := GVL_CAN.ID20_LedBlinkGreen OR DWORD_TO_UINT(BitMask); END_IF
        IF (GVL_CAN.ID20_LedBlue AND DWORD_TO_UINT(BitMask)) > 0 THEN GVL_CAN.ID20_LedBlinkBlue := GVL_CAN.ID20_LedBlinkBlue OR DWORD_TO_UINT(BitMask); END_IF
    END_IF
END_FOR

END_PROGRAM

// ---- POUs/PRG_Ballast.TcPOU
PROGRAM PRG_Ballast
VAR
    // Instanciranje blokova za Port i Stbd
    fbValve_P1, fbValve_P2, fbValve_P3 : FB_BallastValve;
    fbValve_S1, fbValve_S2, fbValve_S3 : FB_BallastValve;
    fbValve_Tunel : FB_BallastValve;
	
	fbTunelPump : FB_TunelPump;
	
	fbScaleP1, fbScaleP2, fbScaleP3 : FB_TankScaling;
	fbScaleS1, fbScaleS2, fbScaleS3 : FB_TankScaling;

    // Triggeri za tipke (CAN + HMI)
    rtModeChange : R_TRIG;
    rtCmdP1, rtCmdP2, rtCmdP3 : R_TRIG;
    rtCmdS1, rtCmdS2, rtCmdS3 : R_TRIG;
    rtCmdTunel : R_TRIG;
    rtCmdPump  : R_TRIG;

    // Lokalne varijable stanja (toggle)
    bCmdOpen_P1, bCmdOpen_P2, bCmdOpen_P3 : BOOL;
    bCmdOpen_S1, bCmdOpen_S2, bCmdOpen_S3 : BOOL;
    bCmdOpen_Tunel  : BOOL;
    bCmdRun_TunelPump : BOOL;
END_VAR



(* ========================================================= *)
(* 1. UPRAVLJANJE MODOM RADA (Tipka 13)                      *)
(* ========================================================= *)
rtModeChange(CLK := GVL_CAN.ID20_Status[13]);

IF rtModeChange.Q THEN
    CASE GVL_HMI.eSystemMode OF
        E_ControlMode.OFF:  GVL_HMI.eSystemMode := E_ControlMode.MAN;
        E_ControlMode.MAN:  GVL_HMI.eSystemMode := E_ControlMode.AUTO;
        E_ControlMode.AUTO: GVL_HMI.eSystemMode := E_ControlMode.OFF;
    END_CASE
END_IF

// Vizualizacija moda na tipki 13
CASE GVL_HMI.eSystemMode OF
    E_ControlMode.OFF:  GVL_CAN.ID20_Config[13].Boja := E_BlinkMarine_Color.OFF;
    E_ControlMode.MAN:  GVL_CAN.ID20_Config[13].Boja := E_BlinkMarine_Color.GREEN;
    E_ControlMode.AUTO: GVL_CAN.ID20_Config[13].Boja := E_BlinkMarine_Color.BLUE;
END_CASE

(* ========================================================= *)
(* 2. OBRADA KOMANDI (Samo u MAN modu)                       *)
(* ========================================================= *)
rtCmdP1(CLK := GVL_CAN.ID20_Status[1]  OR GVL_HMI.bCmdOpen_P1);
rtCmdP2(CLK := GVL_CAN.ID20_Status[6]  OR GVL_HMI.bCmdOpen_P2);
rtCmdP3(CLK := GVL_CAN.ID20_Status[11] OR GVL_HMI.bCmdOpen_P3);
rtCmdS1(CLK := GVL_CAN.ID20_Status[5]  OR GVL_HMI.bCmdOpen_S1);
rtCmdS2(CLK := GVL_CAN.ID20_Status[10] OR GVL_HMI.bCmdOpen_S2);
rtCmdS3(CLK := GVL_CAN.ID20_Status[15] OR GVL_HMI.bCmdOpen_S3);
rtCmdTunel(CLK := GVL_CAN.ID20_Status[12] OR GVL_HMI.bCmdOpen_Tunel);
rtCmdPump(CLK  := GVL_CAN.ID20_Status[14] OR GVL_HMI.bCmdRun_TunelPump);

IF GVL_HMI.eSystemMode = E_ControlMode.MAN THEN
    IF rtCmdP1.Q    THEN bCmdOpen_P1     := NOT bCmdOpen_P1;     END_IF
    IF rtCmdP2.Q    THEN bCmdOpen_P2     := NOT bCmdOpen_P2;     END_IF
    IF rtCmdP3.Q    THEN bCmdOpen_P3     := NOT bCmdOpen_P3;     END_IF
    IF rtCmdS1.Q    THEN bCmdOpen_S1     := NOT bCmdOpen_S1;     END_IF
    IF rtCmdS2.Q    THEN bCmdOpen_S2     := NOT bCmdOpen_S2;     END_IF
    IF rtCmdS3.Q    THEN bCmdOpen_S3     := NOT bCmdOpen_S3;     END_IF
    IF rtCmdTunel.Q THEN bCmdOpen_Tunel  := NOT bCmdOpen_Tunel;  END_IF

    // Toggle logika za pumpu
    IF rtCmdPump.Q THEN bCmdRun_TunelPump := NOT bCmdRun_TunelPump; END_IF

    // Automatsko isključivanje pumpe (kraj vode)
    IF fbTunelPump.bOutResetCmd THEN
        bCmdRun_TunelPump := FALSE;
    END_IF

ELSIF GVL_HMI.eSystemMode = E_ControlMode.OFF THEN
    // U OFF modu sve ugasi
    bCmdOpen_P1 := bCmdOpen_P2 := bCmdOpen_P3 := FALSE;
    bCmdOpen_S1 := bCmdOpen_S2 := bCmdOpen_S3 := FALSE;
    bCmdOpen_Tunel    := FALSE;
    bCmdRun_TunelPump := FALSE;
END_IF

(* ========================================================= *)
(* 3. POZIV FUNKCIJSKIH BLOKOVA                              *)
(* ========================================================= *)

// --- BALAST VENTILI ---
fbValve_P1(bCmdOpen := bCmdOpen_P1, bFbOpen := GVL_IO.DI_BAL_P1_OPEN_FB, bFbClosed := GVL_IO.DI_BAL_P1_CLOSE_FB, bReset := GVL_HMI.bCmdResetAll, bOutSolenoid => GVL_IO.DO_BAL_P1, eState => GVL_HMI.eState_P1, bError => GVL_HMI.bAlarm_P1);
fbValve_P2(bCmdOpen := bCmdOpen_P2, bFbOpen := GVL_IO.DI_BAL_P2_OPEN_FB, bFbClosed := GVL_IO.DI_BAL_P2_CLOSE_FB, bReset := GVL_HMI.bCmdResetAll, bOutSolenoid => GVL_IO.DO_BAL_P2, eState => GVL_HMI.eState_P2, bError => GVL_HMI.bAlarm_P2);
fbValve_P3(bCmdOpen := bCmdOpen_P3, bFbOpen := GVL_IO.DI_BAL_P3_OPEN_FB, bFbClosed := GVL_IO.DI_BAL_P3_CLOSE_FB, bReset := GVL_HMI.bCmdResetAll, bOutSolenoid => GVL_IO.DO_BAL_P3, eState => GVL_HMI.eState_P3, bError => GVL_HMI.bAlarm_P3);

fbValve_S1(bCmdOpen := bCmdOpen_S1, bFbOpen := GVL_IO.DI_BAL_S1_OPEN_FB, bFbClosed := GVL_IO.DI_BAL_S1_CLOSE_FB, bReset := GVL_HMI.bCmdResetAll, bOutSolenoid => GVL_IO.DO_BAL_S1, eState => GVL_HMI.eState_S1, bError => GVL_HMI.bAlarm_S1);
fbValve_S2(bCmdOpen := bCmdOpen_S2, bFbOpen := GVL_IO.DI_BAL_S2_OPEN_FB, bFbClosed := GVL_IO.DI_BAL_S2_CLOSE_FB, bReset := GVL_HMI.bCmdResetAll, bOutSolenoid => GVL_IO.DO_BAL_S2, eState => GVL_HMI.eState_S2, bError => GVL_HMI.bAlarm_S2);
fbValve_S3(bCmdOpen := bCmdOpen_S3, bFbOpen := GVL_IO.DI_BAL_S3_OPEN_FB, bFbClosed := GVL_IO.DI_BAL_S3_CLOSE_FB, bReset := GVL_HMI.bCmdResetAll, bOutSolenoid => GVL_IO.DO_BAL_S3, eState => GVL_HMI.eState_S3, bError => GVL_HMI.bAlarm_S3);

// --- TUNEL VENTIL (Tipka 12) ---
fbValve_Tunel(bCmdOpen := bCmdOpen_Tunel, bFbOpen := GVL_IO.DI_TUNEL_OPEN_FB, bFbClosed := GVL_IO.DI_TUNEL_CLOSE_FB, bReset := GVL_HMI.bCmdResetAll, bOutSolenoid => GVL_IO.DO_TUNEL_VALVE, eState => GVL_HMI.eState_Tunel, bError => GVL_HMI.bAlarm_Tunel);

// --- TUNEL PUMPA (Tipka 14) ---
fbTunelPump(
    bCmdRun      := bCmdRun_TunelPump,
    eValveState  := fbValve_Tunel.eState,
    bSondaPort   := GVL_IO.DI_Sonda_Port,
    bSondaStbd   := GVL_IO.DI_Sonda_Stbd,
    tDryRunDelay := T#6S,
    bClutchOut    => GVL_IO.DO_TunelClutch,
    bSondePowerOut => GVL_IO.DO_SondePower
);

(* ========================================================= *)
(* 4. FEEDBACK NA TIPKOVNICU                                 *)
(* ========================================================= *)

// --- TUNEL VENTIL (Tipka 12) ---
IF fbValve_Tunel.bError THEN 
    GVL_CAN.ID20_Config[12].Boja := E_BlinkMarine_Color.YELLOW; GVL_CAN.ID20_Config[12].Blink := TRUE;
ELSIF fbValve_Tunel.eState = 1 THEN 
    GVL_CAN.ID20_Config[12].Boja := E_BlinkMarine_Color.RED; GVL_CAN.ID20_Config[12].Blink := FALSE;
ELSIF fbValve_Tunel.eState = 2 THEN 
    GVL_CAN.ID20_Config[12].Boja := E_BlinkMarine_Color.GREEN; GVL_CAN.ID20_Config[12].Blink := FALSE;
ELSIF fbValve_Tunel.eState = 0 THEN 
    GVL_CAN.ID20_Config[12].Boja := E_BlinkMarine_Color.YELLOW; GVL_CAN.ID20_Config[12].Blink := FALSE;
ELSE 
    GVL_CAN.ID20_Config[12].Boja := E_BlinkMarine_Color.OFF;
END_IF

// --- TUNEL PUMPA (Tipka 14) ---
IF fbTunelPump.bHasWater THEN
    GVL_CAN.ID20_Config[14].Boja := E_BlinkMarine_Color.BLUE; GVL_CAN.ID20_Config[14].Blink := FALSE;
ELSIF fbTunelPump.bDryRunning THEN
    GVL_CAN.ID20_Config[14].Boja := E_BlinkMarine_Color.YELLOW; GVL_CAN.ID20_Config[14].Blink := TRUE;
ELSE
    // Ako se pumpa sama ugasila (Reset), boja će postati OFF
    GVL_CAN.ID20_Config[14].Boja := E_BlinkMarine_Color.OFF; GVL_CAN.ID20_Config[14].Blink := FALSE;
END_IF

// --- PORT VENTILI (1, 6, 11) ---
// P1
IF fbValve_P1.bError THEN GVL_CAN.ID20_Config[1].Boja := E_BlinkMarine_Color.RED; GVL_CAN.ID20_Config[1].Blink := TRUE;
ELSIF fbValve_P1.eState = 1 THEN GVL_CAN.ID20_Config[1].Boja := E_BlinkMarine_Color.CYAN;
ELSIF fbValve_P1.eState = 2 THEN GVL_CAN.ID20_Config[1].Boja := E_BlinkMarine_Color.GREEN;
ELSIF fbValve_P1.eState = 0 THEN GVL_CAN.ID20_Config[1].Boja := E_BlinkMarine_Color.YELLOW;
ELSE GVL_CAN.ID20_Config[1].Boja := E_BlinkMarine_Color.OFF; END_IF
// P2
IF fbValve_P2.bError THEN GVL_CAN.ID20_Config[6].Boja := E_BlinkMarine_Color.RED; GVL_CAN.ID20_Config[6].Blink := TRUE;
ELSIF fbValve_P2.eState = 1 THEN GVL_CAN.ID20_Config[6].Boja := E_BlinkMarine_Color.CYAN;
ELSIF fbValve_P2.eState = 2 THEN GVL_CAN.ID20_Config[6].Boja := E_BlinkMarine_Color.GREEN;
ELSIF fbValve_P2.eState = 0 THEN GVL_CAN.ID20_Config[6].Boja := E_BlinkMarine_Color.YELLOW;
ELSE GVL_CAN.ID20_Config[6].Boja := E_BlinkMarine_Color.OFF; END_IF
// P3
IF fbValve_P3.bError THEN GVL_CAN.ID20_Config[11].Boja := E_BlinkMarine_Color.RED; GVL_CAN.ID20_Config[11].Blink := TRUE;
ELSIF fbValve_P3.eState = 1 THEN GVL_CAN.ID20_Config[11].Boja := E_BlinkMarine_Color.CYAN;
ELSIF fbValve_P3.eState = 2 THEN GVL_CAN.ID20_Config[11].Boja := E_BlinkMarine_Color.GREEN;
ELSIF fbValve_P3.eState = 0 THEN GVL_CAN.ID20_Config[11].Boja := E_BlinkMarine_Color.YELLOW;
ELSE GVL_CAN.ID20_Config[11].Boja := E_BlinkMarine_Color.OFF; END_IF

// --- STBD VENTILI (5, 10, 15) ---
// S1
IF fbValve_S1.bError THEN GVL_CAN.ID20_Config[5].Boja := E_BlinkMarine_Color.RED; GVL_CAN.ID20_Config[5].Blink := TRUE;
ELSIF fbValve_S1.eState = 1 THEN GVL_CAN.ID20_Config[5].Boja := E_BlinkMarine_Color.CYAN;
ELSIF fbValve_S1.eState = 2 THEN GVL_CAN.ID20_Config[5].Boja := E_BlinkMarine_Color.GREEN;
ELSIF fbValve_S1.eState = 0 THEN GVL_CAN.ID20_Config[5].Boja := E_BlinkMarine_Color.YELLOW;
ELSE GVL_CAN.ID20_Config[5].Boja := E_BlinkMarine_Color.OFF; END_IF
// S2
IF fbValve_S2.bError THEN GVL_CAN.ID20_Config[10].Boja := E_BlinkMarine_Color.RED; GVL_CAN.ID20_Config[10].Blink := TRUE;
ELSIF fbValve_S2.eState = 1 THEN GVL_CAN.ID20_Config[10].Boja := E_BlinkMarine_Color.CYAN;
ELSIF fbValve_S2.eState = 2 THEN GVL_CAN.ID20_Config[10].Boja := E_BlinkMarine_Color.GREEN;
ELSIF fbValve_S2.eState = 0 THEN GVL_CAN.ID20_Config[10].Boja := E_BlinkMarine_Color.YELLOW;
ELSE GVL_CAN.ID20_Config[10].Boja := E_BlinkMarine_Color.OFF; END_IF
// S3
IF fbValve_S3.bError THEN GVL_CAN.ID20_Config[15].Boja := E_BlinkMarine_Color.RED; GVL_CAN.ID20_Config[15].Blink := TRUE;
ELSIF fbValve_S3.eState = 1 THEN GVL_CAN.ID20_Config[15].Boja := E_BlinkMarine_Color.CYAN;
ELSIF fbValve_S3.eState = 2 THEN GVL_CAN.ID20_Config[15].Boja := E_BlinkMarine_Color.GREEN;
ELSIF fbValve_S3.eState = 0 THEN GVL_CAN.ID20_Config[15].Boja := E_BlinkMarine_Color.YELLOW;
ELSE GVL_CAN.ID20_Config[15].Boja := E_BlinkMarine_Color.OFF; END_IF

(* ========================================================= *)
(* 5. SKALIRANJE NIVOA TANKOVA (HMI I DISPLAY)               *)
(* ========================================================= *)

// PORT TANKOVI
fbScaleP1(
    iRawIn  := GVL_IO.iLevel_Bal_P1_Raw, 
    iInMin  := 4553, iInMax := 32767, 
    iOutMin := 4553, iOutMax := 32767, 
    fPercentage => GVL_IO.fLevel_Bal_P1_Pct_Hmi, 
    iRawOut => GVL_IO.fLevel_Bal_P1_Pct_Disp);

fbScaleP2(
    iRawIn  := GVL_IO.iLevel_Bal_P2_Raw, 
    iInMin  := 4553, iInMax := 32767, 
    iOutMin := 4553, iOutMax := 32767, 
    fPercentage => GVL_IO.fLevel_Bal_P2_Pct_Hmi, 
    iRawOut => GVL_IO.fLevel_Bal_P2_Pct_Disp);

fbScaleP3(
    iRawIn  := GVL_IO.iLevel_Bal_P3_Raw, 
    iInMin  := 4553, iInMax := 32767, 
    iOutMin := 4553, iOutMax := 32767, 
    fPercentage => GVL_IO.fLevel_Bal_P3_Pct_Hmi, 
    iRawOut => GVL_IO.fLevel_Bal_P3_Pct_Disp);

// STBD TANKOVI
fbScaleS1(
    iRawIn  := GVL_IO.iLevel_Bal_S1_Raw, 
    iInMin  := 4553, iInMax := 32767, 
    iOutMin := 4553, iOutMax := 32767, 
    fPercentage => GVL_IO.fLevel_Bal_S1_Pct_Hmi, 
    iRawOut => GVL_IO.fLevel_Bal_S1_Pct_Disp);

fbScaleS2(
    iRawIn  := GVL_IO.iLevel_Bal_S2_Raw, 
    iInMin  := 4553, iInMax := 32767, 
    iOutMin := 4553, iOutMax := 32767, 
    fPercentage => GVL_IO.fLevel_Bal_S2_Pct_Hmi, 
    iRawOut => GVL_IO.fLevel_Bal_S2_Pct_Disp);

fbScaleS3(
    iRawIn  := GVL_IO.iLevel_Bal_S3_Raw, 
    iInMin  := 0, iInMax := 32767, 
    iOutMin := 0, iOutMax := 32767, 
    fPercentage => GVL_IO.fLevel_Bal_S3_Pct_Hmi, 
    iRawOut => GVL_IO.fLevel_Bal_S3_Pct_Disp);

END_PROGRAM

// ---- POUs/FBs/FB_BallastValve.TcPOU
FUNCTION_BLOCK FB_BallastValve
VAR_INPUT
    bCmdOpen   : BOOL;       (* TRUE = Otvori, FALSE = Zatvori *)
    bFbOpen    : BOOL;       (* Feedback senzor: Otvoren *)
    bFbClosed  : BOOL;       (* Feedback senzor: Zatvoren *)
    bReset     : BOOL;       (* Reset alarma *)
    tTimeout   : TIME := T#3S; (* Vrijeme za timeout, default 3s *)
END_VAR

VAR_OUTPUT
    bOutSolenoid : BOOL;         (* Izlaz na špulu *)
    eState       : E_ValveState; (* Trenutno stanje za logiku/HMI *)
    bError       : BOOL;         (* Zbirna greška *)
    bErrTimeout  : BOOL;         (* Greška: Nije stigao na vrijeme *)
    bErrSensor   : BOOL;         (* Greška: Oba senzora aktivna *)
END_VAR

VAR
    tmrMove      : TON;          (* Timer za praćenje kretanja *)
    rtCmdOpen    : R_TRIG;       (* Rastući brid - komanda "Otvori" *)
    ftCmdClose   : F_TRIG;       (* Padajući brid - komanda "Zatvori" *)
    bCmdActive   : BOOL;         (* TRUE tek kad je komanda aktivno dana, sprječava lažni timeout pri PowerOn *)
END_VAR

// 1. Upravljanje fizičkim izlazom (Solenoid)
bOutSolenoid := bCmdOpen;

// 2. Evaluacija stanja ventila na temelju senzora
// Mapiranje: 0=Unknown, 1=Open, 2=Closed, 3=Error

IF bFbOpen AND NOT bFbClosed THEN
    eState := 1; // VALVE_OPEN
    bErrSensor := FALSE; 
    
ELSIF NOT bFbOpen AND bFbClosed THEN
    eState := 2; // VALVE_CLOSED
    bErrSensor := FALSE;

ELSIF bFbOpen AND bFbClosed THEN
    eState := 3; // VALVE_ERROR
    bErrSensor := TRUE; // Nemoguće stanje (oba senzora aktivna)

ELSE
    eState := 0; // VALVE_UNKNOWN (Niti jedan senzor - u putovanju)
END_IF

// 3. Detekcija nove komande (timer se aktivira tek na promjenu komande, ne pri PowerOn)
rtCmdOpen(CLK := bCmdOpen);
ftCmdClose(CLK := bCmdOpen);

IF rtCmdOpen.Q OR ftCmdClose.Q THEN
    bCmdActive := TRUE;
END_IF

// 4. Logika Timeout-a (samo ako je komanda aktivno dana)
IF bCmdActive THEN
    IF (bCmdOpen AND eState = 1) OR (NOT bCmdOpen AND eState = 2) THEN
        bCmdActive := FALSE; // Cilj dostignut, zaustavi timer
    END_IF
END_IF

tmrMove(IN := bCmdActive, PT := tTimeout);

// 5. Postavljanje Timeout greške
IF tmrMove.Q THEN
    bErrTimeout := TRUE;
    bCmdActive  := FALSE; // Zaustavi timer nakon greške
END_IF

// 6. Resetiranje grešaka
IF bReset THEN
    bErrTimeout := FALSE;
    bErrSensor  := FALSE;
    bCmdActive  := FALSE; // Reset komande — korisnik mora ponovo dati komandu
END_IF

// 6. Zbirni izlaz za grešku
bError := bErrTimeout OR bErrSensor;

END_FUNCTION_BLOCK

// ---- POUs/FBs/FB_TunelPump.TcPOU
FUNCTION_BLOCK FB_TunelPump
VAR_INPUT
    bCmdRun        : BOOL;    
    eValveState    : INT;     
    bSondaPort     : BOOL;    
    bSondaStbd     : BOOL;    
    tDryRunDelay   : TIME := T#6S; 
END_VAR

VAR_OUTPUT
    bClutchOut     : BOOL;    
    bSondePowerOut : BOOL;    
    bHasWater      : BOOL;    
    bDryRunning    : BOOL;    
    bOutResetCmd   : BOOL; // NOVO: Izlaz za automatsko resetiranje komande
END_VAR

VAR
    tmrDryRun      : TON;     
    bActiveSonda   : BOOL;    
END_VAR

// 1. Odabir aktivne sonde
IF eValveState = 1 THEN
    bActiveSonda := bSondaPort;
ELSIF eValveState = 2 THEN
    bActiveSonda := bSondaStbd;
ELSE
    bActiveSonda := FALSE;
END_IF

// 2. Logika rada i Dry-Run tajmera
tmrDryRun(IN := bCmdRun AND NOT bActiveSonda, PT := tDryRunDelay);

// Ako tajmer odradi (suhi rad), šaljemo impuls za reset
bOutResetCmd := tmrDryRun.Q;

// Pumpa radi samo ako NIJE aktivan tajmer suhog rada
IF bCmdRun AND NOT tmrDryRun.Q THEN
    bClutchOut := TRUE;
ELSE
    bClutchOut := FALSE;
END_IF

bSondePowerOut := bClutchOut;

// 3. Statusi za vizualizaciju
bHasWater    := bClutchOut AND bActiveSonda;
bDryRunning  := bClutchOut AND NOT bActiveSonda;

END_FUNCTION_BLOCK

// ---- POUs/FBs/FB_TankScaling.TcPOU
FUNCTION_BLOCK FB_TankScaling
VAR_INPUT
    iRawIn          : INT;          (* Sirova vrijednost s AI kartice (4-20mA) *)
    iInMin          : INT := 0;     (* Npr. 0 ili 4000 ovisno o senzoru *)
    iInMax          : INT := 32767;
    iOutMin         : INT := 0;     (* Vrijednost za AO EL4018 na 4mA *)
    iOutMax         : INT := 32767; (* Vrijednost za AO EL4018 na 20mA *)
END_VAR
VAR_OUTPUT
    fPercentage     : REAL;         (* 0.0 - 100.0 % za HMI *)
    iRawOut         : INT;          (* Izlaz za Display (AO kartica) *)
END_VAR
VAR
    fTemp           : REAL;
END_VAR

// 1. Izračun postotka (Input Scaling)
IF (iInMax - iInMin) <> 0 THEN
    fTemp := (INT_TO_REAL(iRawIn) - INT_TO_REAL(iInMin)) / (INT_TO_REAL(iInMax) - INT_TO_REAL(iInMin));
    fPercentage := LIMIT(0.0, fTemp * 100.0, 100.0);
ELSE
    fPercentage := 0.0;
END_IF

// 2. Izračun izlaza za Display (Output Scaling)
// fPercentage (0-100) skaliramo na opseg iOutMin do iOutMax
iRawOut := REAL_TO_INT((fPercentage / 100.0) * INT_TO_REAL(iOutMax - iOutMin) + INT_TO_REAL(iOutMin));

END_FUNCTION_BLOCK

// ---- POUs/PRG_Doors.TcPOU

PROGRAM PRG_Doors
VAR
    (* Instance kontrolnih blokova za vrata *)
    fbDoorFwd : FB_DoorControl;
    fbDoorAft : FB_DoorControl;

    (* Triggeri za tipke na tipkovnici *)
    rtBtnDoorFwd : R_TRIG;
    rtBtnDoorAft : R_TRIG;

    (* Drive mode *)
    eTargetMode  : E_SystemMode := E_SystemMode.MODE_IDLE;
    bTurbineSafe : BOOL;

    (* Triggeri za Tipku 4 s obje tipkovnice *)
    rtMode_ID10 : R_TRIG;
    rtMode_ID11 : R_TRIG;

    (* Edge detekcija za ulaz/izlaz iz DRIVE *)
    rtDriveOn  : R_TRIG;
    rtDriveOff : F_TRIG;

    (* 0 = nema sekvence, 1 = otvaranje, 2 = zatvaranje *)
    iDoorSeq : INT := 0;

    (* Reset vrata *)
    bResetDoors : BOOL := FALSE;
END_VAR


// =========================================================
// 1. KONTROLA MODA (Tipka 4)
// =========================================================
bTurbineSafe := (GVL_IO.fEngineRPM_Scaled < 900.0);

rtMode_ID10(CLK := GVL_CAN.ID10_Status[4]);
rtMode_ID11(CLK := GVL_CAN.ID11_Status[4]);

IF bTurbineSafe AND (rtMode_ID10.Q OR rtMode_ID11.Q) THEN
    IF eTargetMode = E_SystemMode.MODE_IDLE THEN
        eTargetMode := E_SystemMode.MODE_DRIVE;
    ELSE
        eTargetMode := E_SystemMode.MODE_IDLE;
    END_IF
END_IF;

// Rubovi DRIVE moda
rtDriveOn(CLK := (eTargetMode = E_SystemMode.MODE_DRIVE));
rtDriveOff(CLK := (eTargetMode = E_SystemMode.MODE_DRIVE));


// =========================================================
// 2. POKRETANJE SEKVENCI
// =========================================================
// Ulaz u DRIVE -> pokreni sekvencu otvaranja
IF rtDriveOn.Q THEN
    iDoorSeq := 1;
END_IF;

// Izlaz iz DRIVE -> pokreni sekvencu zatvaranja
IF rtDriveOff.Q THEN
    iDoorSeq := 2;
END_IF;


// =========================================================
// 3. DEFAULT KOMANDE
// =========================================================
GVL_HMI.bCmdDoorFwd_Open := FALSE;
GVL_HMI.bCmdDoorFwd_Close := FALSE;
GVL_HMI.bCmdDoorAft_Open := FALSE;
GVL_HMI.bCmdDoorAft_Close := FALSE;


// =========================================================
// 4. RUČNI RAD SAMO KAD NEMA DRIVE SEKVENCE
//    I KAD NIJE AKTIVAN DRIVE MODE
// =========================================================
IF (iDoorSeq = 0) AND (eTargetMode <> E_SystemMode.MODE_DRIVE) THEN
    rtBtnDoorFwd(CLK := GVL_CAN.ID20_Status[3] OR GVL_HMI.bCmdDoorFwd);
    rtBtnDoorAft(CLK := GVL_CAN.ID20_Status[8] OR GVL_HMI.bCmdDoorAft);

    IF GVL_HMI.eSystemMode = E_ControlMode.MAN THEN

        IF rtBtnDoorFwd.Q THEN
            IF (fbDoorFwd.eState = E_DoorState.OPEN) OR (fbDoorFwd.eState = E_DoorState.TRAVELING_OPEN) THEN
                GVL_HMI.bCmdDoorFwd_Open := FALSE;
                GVL_HMI.bCmdDoorFwd_Close := TRUE;
            ELSE
                GVL_HMI.bCmdDoorFwd_Open := TRUE;
                GVL_HMI.bCmdDoorFwd_Close := FALSE;
            END_IF
        END_IF

        IF rtBtnDoorAft.Q THEN
            IF (fbDoorAft.eState = E_DoorState.OPEN) OR (fbDoorAft.eState = E_DoorState.TRAVELING_OPEN) THEN
                GVL_HMI.bCmdDoorAft_Open := FALSE;
                GVL_HMI.bCmdDoorAft_Close := TRUE;
            ELSE
                GVL_HMI.bCmdDoorAft_Open := TRUE;
                GVL_HMI.bCmdDoorAft_Close := FALSE;
            END_IF
        END_IF

    ELSIF GVL_HMI.eSystemMode = E_ControlMode.OFF THEN
        // sve ostaje FALSE
    END_IF
END_IF;


// =========================================================
// 5. SEKVENCA VRATA
//    1 = OTVARANJE FWD -> AFT
//    2 = ZATVARANJE FWD -> AFT
// =========================================================
CASE iDoorSeq OF

    0:
        // nema sekvence

    1: // OTVARANJE
        // prvo FWD, pa kad je otvoren onda AFT
        IF fbDoorFwd.eState <> E_DoorState.OPEN THEN
            GVL_HMI.bCmdDoorFwd_Open := TRUE;
            GVL_HMI.bCmdDoorFwd_Close := FALSE;

            GVL_HMI.bCmdDoorAft_Open := FALSE;
            GVL_HMI.bCmdDoorAft_Close := FALSE;

        ELSIF fbDoorAft.eState <> E_DoorState.OPEN THEN
            GVL_HMI.bCmdDoorFwd_Open := FALSE;
            GVL_HMI.bCmdDoorFwd_Close := FALSE;

            GVL_HMI.bCmdDoorAft_Open := TRUE;
            GVL_HMI.bCmdDoorAft_Close := FALSE;

        ELSE
            // oba otvorena -> sekvenca gotova
            iDoorSeq := 0;
        END_IF


    2: // ZATVARANJE
        // prvo FWD, pa kad je zatvoren onda AFT
        IF fbDoorFwd.eState <> E_DoorState.CLOSED THEN
            GVL_HMI.bCmdDoorFwd_Open := FALSE;
            GVL_HMI.bCmdDoorFwd_Close := TRUE;

            GVL_HMI.bCmdDoorAft_Open := FALSE;
            GVL_HMI.bCmdDoorAft_Close := FALSE;

        ELSIF fbDoorAft.eState <> E_DoorState.CLOSED THEN
            GVL_HMI.bCmdDoorFwd_Open := FALSE;
            GVL_HMI.bCmdDoorFwd_Close := FALSE;

            GVL_HMI.bCmdDoorAft_Open := FALSE;
            GVL_HMI.bCmdDoorAft_Close := TRUE;

        ELSE
            // oba zatvorena -> sekvenca gotova
            iDoorSeq := 0;
        END_IF


ELSE
    iDoorSeq := 0;
END_CASE;


// =========================================================
// 6. POZIV FB BLOKOVA
// =========================================================
fbDoorFwd(
    bCmdOpen := GVL_HMI.bCmdDoorFwd_Open,
    bCmdClose := GVL_HMI.bCmdDoorFwd_Close,
    bReset := bResetDoors,
    bEnableRefill := TRUE,
    fPresOpen := GVL_IO.fPressure_FWD_A,
    fPresClose := GVL_IO.fPressure_FWD_B,
    fLimitOpen := 60.0,
    fLimitClose := 60.0,
    bSolOpen => GVL_IO.DO_DoorFwd_Open,
    bSolClose => GVL_IO.DO_DoorFwd_Close,
    eState => GVL_HMI.eState_DoorFwd
);

fbDoorAft(
    bCmdOpen := GVL_HMI.bCmdDoorAft_Open,
    bCmdClose := GVL_HMI.bCmdDoorAft_Close,
    bReset := bResetDoors,
    bEnableRefill := TRUE,
    fPresOpen := GVL_IO.fPressure_AFT_A,
    fPresClose := GVL_IO.fPressure_AFT_B,
    fLimitOpen := 60.0,
    fLimitClose := 60.0,
    bSolOpen => GVL_IO.DO_DoorAft_Open,
    bSolClose => GVL_IO.DO_DoorAft_Close,
    eState => GVL_HMI.eState_DoorAft
);


// =========================================================
// 7. INDIKACIJA MODA
// =========================================================
IF eTargetMode = E_SystemMode.MODE_DRIVE THEN
    GVL_CAN.ID10_Config[4].Boja := E_BlinkMarine_Color.GREEN;
    GVL_CAN.ID11_Config[4].Boja := E_BlinkMarine_Color.GREEN;
ELSE
    GVL_CAN.ID10_Config[4].Boja := E_BlinkMarine_Color.OFF;
    GVL_CAN.ID11_Config[4].Boja := E_BlinkMarine_Color.OFF;
END_IF;


// =========================================================
// 8. INDIKACIJA STANJA VRATA NA ID20
// =========================================================

// FWD (Tipka 3)
// Solid: CYAN=Otvoreno, GREEN=Zatvoreno | Blink: CYAN=Putuje prema otvorenom, GREEN=Putuje prema zatvorenom
IF fbDoorFwd.eState = E_DoorState.OPEN THEN
    GVL_CAN.ID20_Config[3].Boja  := E_BlinkMarine_Color.CYAN;
    GVL_CAN.ID20_Config[3].Blink := FALSE;
ELSIF fbDoorFwd.eState = E_DoorState.CLOSED THEN
    GVL_CAN.ID20_Config[3].Boja  := E_BlinkMarine_Color.GREEN;
    GVL_CAN.ID20_Config[3].Blink := FALSE;
ELSIF fbDoorFwd.eState = E_DoorState.TRAVELING_OPEN THEN
    GVL_CAN.ID20_Config[3].Boja  := E_BlinkMarine_Color.CYAN;
    GVL_CAN.ID20_Config[3].Blink := TRUE;
ELSIF fbDoorFwd.eState = E_DoorState.TRAVELING_CLOSE THEN
    GVL_CAN.ID20_Config[3].Boja  := E_BlinkMarine_Color.GREEN;
    GVL_CAN.ID20_Config[3].Blink := TRUE;
ELSE
    GVL_CAN.ID20_Config[3].Boja  := E_BlinkMarine_Color.OFF;
    GVL_CAN.ID20_Config[3].Blink := FALSE;
END_IF;

// AFT (Tipka 8)
IF fbDoorAft.eState = E_DoorState.OPEN THEN
    GVL_CAN.ID20_Config[8].Boja  := E_BlinkMarine_Color.CYAN;
    GVL_CAN.ID20_Config[8].Blink := FALSE;
ELSIF fbDoorAft.eState = E_DoorState.CLOSED THEN
    GVL_CAN.ID20_Config[8].Boja  := E_BlinkMarine_Color.GREEN;
    GVL_CAN.ID20_Config[8].Blink := FALSE;
ELSIF fbDoorAft.eState = E_DoorState.TRAVELING_OPEN THEN
    GVL_CAN.ID20_Config[8].Boja  := E_BlinkMarine_Color.CYAN;
    GVL_CAN.ID20_Config[8].Blink := TRUE;
ELSIF fbDoorAft.eState = E_DoorState.TRAVELING_CLOSE THEN
    GVL_CAN.ID20_Config[8].Boja  := E_BlinkMarine_Color.GREEN;
    GVL_CAN.ID20_Config[8].Blink := TRUE;
ELSE
    GVL_CAN.ID20_Config[8].Boja  := E_BlinkMarine_Color.OFF;
    GVL_CAN.ID20_Config[8].Blink := FALSE;
END_IF;

END_PROGRAM

// ---- POUs/FBs/FB_DoorControl.TcPOU
FUNCTION_BLOCK FB_DoorControl
VAR_INPUT
    bCmdOpen      : BOOL;
    bCmdClose     : BOOL;
    bReset        : BOOL;
    bEnableRefill : BOOL := TRUE;
    fPresOpen     : REAL;
    fPresClose    : REAL;
    fLimitOpen    : REAL := 50.0;
    fLimitClose   : REAL := 120.0;
    fHysteresis   : REAL := 15.0;
    tTimeout      : TIME := T#15S;
    tRefillMax    : TIME := T#6S;
END_VAR

VAR_OUTPUT
    bSolOpen      : BOOL;
    bSolClose     : BOOL;
    eState        : E_DoorState;
    bError        : BOOL;
    bLeakAlarm    : BOOL;
END_VAR

VAR
    tmrMove       : TON;
    tmrRefill     : TON;
    bRefilling    : BOOL := FALSE;
    iInternalSt   : INT := 0;

    fStartOpen    : REAL;
    fStopOpen     : REAL;
    fStartClose   : REAL;
    fStopClose    : REAL;
END_VAR


// 1. RESET
IF bReset THEN
    bError := FALSE;
    bLeakAlarm := FALSE;
    bRefilling := FALSE;
    iInternalSt := 0;

    bSolOpen := FALSE;
    bSolClose := FALSE;
    eState := E_DoorState.IDLE;

    tmrMove(IN := FALSE, PT := tTimeout);
    tmrRefill(IN := FALSE, PT := tRefillMax);
    RETURN;
END_IF;

// NAPOMENA: bError i bLeakAlarm su SAMO indikacije (HMI alarm).
// Sustav namjerno NE zaustavlja rad vrata na alarm — operater odlučuje.

// 2. STATE MACHINE
CASE iInternalSt OF

    0: // IDLE
        bSolOpen := FALSE;
        bSolClose := FALSE;
        bRefilling := FALSE;
        eState := E_DoorState.IDLE;

        IF bCmdOpen AND NOT bCmdClose THEN
            bError      := FALSE; // Nova komanda čisti prethodnu timeout grešku
            iInternalSt := 10;
        ELSIF bCmdClose AND NOT bCmdOpen THEN
            bError      := FALSE;
            iInternalSt := 20;
        END_IF


    10: // PUTOVANJE OTVARANJE
        bSolOpen := TRUE;
        bSolClose := FALSE;
        bRefilling := FALSE;
        eState := E_DoorState.TRAVELING_OPEN;

        IF fPresOpen >= fLimitOpen THEN
            iInternalSt := 1;
        ELSIF bCmdClose THEN
            iInternalSt := 20;
        END_IF


    1: // OTVORENO - ODRŽAVANJE TLAKA
        bSolClose := FALSE;
        eState := E_DoorState.OPEN;

        IF bEnableRefill THEN
            IF fPresOpen <= (fLimitOpen - fHysteresis) THEN
                bRefilling := TRUE;
            ELSIF fPresOpen >= fLimitOpen THEN
                bRefilling := FALSE;
            END_IF
        ELSE
            bRefilling := FALSE;
        END_IF

        bSolOpen := bRefilling;

        IF bCmdClose AND NOT bCmdOpen THEN
            bRefilling := FALSE;
            iInternalSt := 20;
        END_IF


    20: // PUTOVANJE ZATVARANJE
        bSolOpen := FALSE;
        bSolClose := TRUE;
        bRefilling := FALSE;
        eState := E_DoorState.TRAVELING_CLOSE;

        IF fPresClose >= fLimitClose THEN
            iInternalSt := 2;
        ELSIF bCmdOpen THEN
            iInternalSt := 10;
        END_IF


    2: // ZATVORENO - ODRŽAVANJE TLAKA
        bSolOpen := FALSE;
        eState := E_DoorState.CLOSED;

        IF bEnableRefill THEN
            IF fPresClose <= (fLimitClose - fHysteresis) THEN
                bRefilling := TRUE;
            ELSIF fPresClose >= fLimitClose THEN
                bRefilling := FALSE;
            END_IF
        ELSE
            bRefilling := FALSE;
        END_IF

        bSolClose := bRefilling;

        IF bCmdOpen AND NOT bCmdClose THEN
            bRefilling := FALSE;
            iInternalSt := 10;
        END_IF


ELSE
    bSolOpen := FALSE;
    bSolClose := FALSE;
    bRefilling := FALSE;
    eState := E_DoorState.IDLE;
    iInternalSt := 0;
END_CASE


// 4. TIMERI
tmrMove(IN := (iInternalSt = 10) OR (iInternalSt = 20), PT := tTimeout);
IF tmrMove.Q THEN
    bError       := TRUE;
    iInternalSt  := 0; // Vrati u IDLE — isključi solenoid, čekaj reset od operatera
END_IF

tmrRefill(IN := bRefilling, PT := tRefillMax);
IF tmrRefill.Q THEN
    bLeakAlarm := TRUE;
END_IF

END_FUNCTION_BLOCK

// ---- POUs/PRG_Winches.TcPOU
PROGRAM PRG_Winches
VAR
    (* --- INSTANCE KONTROLNIH BLOKOVA --- *)
    fbWinch1 : FB_WinchControl;
    fbWinch2 : FB_WinchControl;
    fbWinch3 : FB_WinchControl;

    (* --- HMI STRUKTURE --- *)
    // Ove strukture linkaš na svoj HMI ekran za ručno upravljanje i animacije
    stWinch1_HMI : ST_UcWinchControl;
    stWinch2_HMI : ST_UcWinchControl;
    stWinch3_HMI : ST_UcWinchControl;

    (* --- INTERNE VARIJABLE --- *)
    iActiveCount : INT := 0;
    iRpmPerWinch : INT := 200; 
    iBaseRpm     : INT := 700; 
    
    tmrDCPumpOff : TOF; // Timer za gašenje DC pumpe
    bEngineIsOn  : BOOL;
    
    // Glavna dozvola za rad vinčeva — AND oba NC stop prekidača
    bSystemSafe  : BOOL;
END_VAR

